KUKA KRL program: MyProgram_200().src

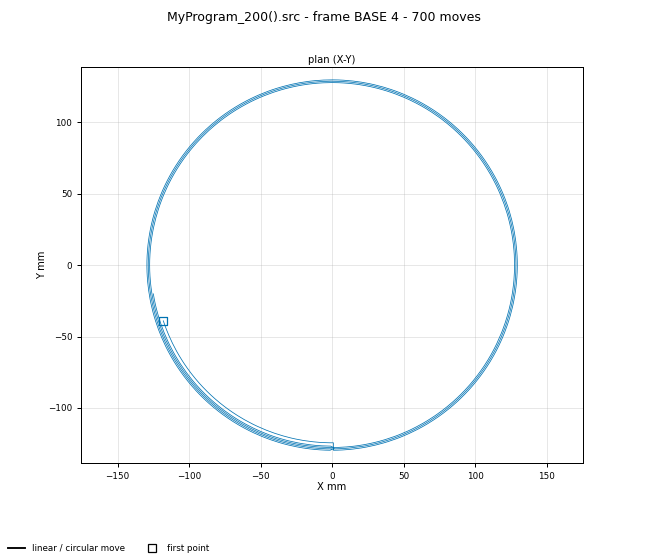
[picture p0: tool path of MyProgram_200().src in frame BASE 4, 700 of 700 moves have a stored position in this frame; points joined in program order, loops and branches not executed]
&ACCESS RVP
&REL 1
&PARAM TEMPLATE = C:\KRC\Roboter\Template\vorgabe
&PARAM EDITMASK = *
DEF MyProgram_200()
; ---- Setting reference (Base) ----
$BASE = BASE_DATA[4]

; --------------------------
; ---- Setting tool (TCP) ----
$TOOL = TOOL_DATA[3]
; --------------------------

$VEL.CP = VEL_APROX_PRINT
Startdeposition()
$VEL.CP = VEL_PRINT
LIN {X -118.0723,Y -39.0089,Z 143,A -163.9412,B 21.6303,C -0.9497,E1 21.4984,E2 611.217} C_DIS
LIN {X -116.9975,Y -42.1221,Z 143,A -162.4124,B 21.6305,C -0.9457,E1 21.4998,E2 609.6889} C_DIS
LIN {X -115.7317,Y -45.4869,Z 143,A -160.5818,B 21.6305,C -0.9476,E1 21.5017,E2 607.8411} C_DIS
LIN {X -114.1935,Y -49.2192,Z 143,A -158.8658,B 21.6309,C -0.9367,E1 21.5035,E2 606.1436} C_DIS
LIN {X -112.9502,Y -52.0092,Z 143,A -157.5422,B 21.6312,C -0.9295,E1 21.5051,E2 604.831} C_DIS
LIN {X -111.6598,Y -54.7252,Z 143,A -155.9756,B 21.631,C -0.9327,E1 21.507,E2 603.2459} C_DIS
LIN {X -110.264,Y -57.486,Z 143,A -154.672,B 21.6314,C -0.9241,E1 21.5086,E2 601.9576} C_DIS
LIN {X -108.8242,Y -60.1699,Z 143,A -153.2851,B 21.6316,C -0.9196,E1 21.5105,E2 600.5743} C_DIS
LIN {X -107.0458,Y -63.2806,Z 143,A -151.5187,B 21.6316,C -0.9197,E1 21.513,E2 598.7968} C_DIS
LIN {X -104.9264,Y -66.736,Z 143,A -149.6994,B 21.6318,C -0.913,E1 21.5156,E2 596.9849} C_DIS
LIN {X -103.3886,Y -69.0936,Z 143,A -148.3196,B 21.6318,C -0.913,E1 21.5178,E2 595.5972} C_DIS
LIN {X -101.1506,Y -72.3303,Z 143,A -146.4144,B 21.6318,C -0.912,E1 21.5208,E2 593.6835} C_DIS
LIN {X -98.5052,Y -75.8944,Z 143,A -144.3224,B 21.632,C -0.9089,E1 21.5244,E2 591.5883} C_DIS
LIN {X -95.4814,Y -79.6651,Z 143,A -142.1236,B 21.6323,C -0.9026,E1 21.5283,E2 589.3946} C_DIS
LIN {X -92.7275,Y -82.8538,Z 143,A -140.2642,B 21.6326,C -0.895,E1 21.5317,E2 587.5462} C_DIS
LIN {X -90.4998,Y -85.2814,Z 143,A -138.6409,B 21.6326,C -0.8958,E1 21.5348,E2 585.9122} C_DIS
LIN {X -87.3908,Y -88.4652,Z 143,A -136.6816,B 21.6328,C -0.8878,E1 21.5386,E2 583.9648} C_DIS
LIN {X -84.5496,Y -91.1842,Z 143,A -134.7498,B 21.6328,C -0.8889,E1 21.5425,E2 582.0209} C_DIS
LIN {X -81.7041,Y -93.7421,Z 143,A -132.9762,B 21.6329,C -0.8859,E1 21.5463,E2 580.2472} C_DIS
LIN {X -78.2894,Y -96.6125,Z 143,A -130.895,B 21.633,C -0.8831,E1 21.5507,E2 578.1644} C_DIS
LIN {X -75.1041,Y -99.1088,Z 143,A -129.1612,B 21.6334,C -0.8745,E1 21.5545,E2 576.4465} C_DIS
LIN {X -72.66,Y -100.9148,Z 143,A -127.794,B 21.6334,C -0.8708,E1 21.5576,E2 575.0838} C_DIS
LIN {X -69.8722,Y -102.8642,Z 143,A -126.1244,B 21.6334,C -0.8723,E1 21.5615,E2 573.4034} C_DIS
LIN {X -66.3215,Y -105.1883,Z 143,A -124.2918,B 21.6337,C -0.8644,E1 21.5658,E2 571.5855} C_DIS
LIN {X -63.9198,Y -106.6652,Z 143,A -122.8675,B 21.6337,C -0.8675,E1 21.5692,E2 570.1476} C_DIS
LIN {X -61.2916,Y -108.1971,Z 143,A -121.5152,B 21.6337,C -0.8635,E1 21.5724,E2 568.8014} C_DIS
LIN {X -58.1603,Y -109.9099,Z 143,A -119.9844,B 21.634,C -0.8567,E1 21.5762,E2 567.2839} C_DIS
LIN {X -55.5007,Y -111.2772,Z 143,A -118.5783,B 21.634,C -0.8561,E1 21.5797,E2 565.875} C_DIS
LIN {X -52.295,Y -112.818,Z 143,A -116.7434,B 21.6338,C -0.8622,E1 21.5844,E2 564.0183} C_DIS
LIN {X -48.773,Y -114.3864,Z 143,A -115.0584,B 21.634,C -0.8565,E1 21.5887,E2 562.344} C_DIS
LIN {X -46.1695,Y -115.4607,Z 143,A -113.7595,B 21.634,C -0.8553,E1 21.592,E2 561.045} C_DIS
LIN {X -42.8553,Y -116.7331,Z 143,A -112.1391,B 21.6342,C -0.8531,E1 21.5962,E2 559.4267} C_DIS
LIN {X -40.2291,Y -117.663,Z 143,A -110.8366,B 21.6342,C -0.8528,E1 21.5997,E2 558.1221} C_DIS
LIN {X -37.3375,Y -118.6123,Z 143,A -109.4335,B 21.6342,C -0.8517,E1 21.6034,E2 556.7188} C_DIS
LIN {X -34.4074,Y -119.4953,Z 143,A -107.8623,B 21.634,C -0.8574,E1 21.6077,E2 555.1293} C_DIS
LIN {X -31.4493,Y -120.308,Z 143,A -106.6081,B 21.6343,C -0.8499,E1 21.611,E2 553.8931} C_DIS
LIN {X -28.7309,Y -120.9852,Z 143,A -105.1465,B 21.634,C -0.8563,E1 21.615,E2 552.4119} C_DIS
LIN {X -25.5148,Y -121.7056,Z 143,A -103.8017,B 21.6343,C -0.8483,E1 21.6187,E2 551.0867} C_DIS
LIN {X -22.5042,Y -122.2974,Z 143,A -102.4392,B 21.6344,C -0.8457,E1 21.6224,E2 549.7297} C_DIS
LIN {X -19.7621,Y -122.7709,Z 143,A -100.9999,B 21.6342,C -0.8518,E1 21.6264,E2 548.2723} C_DIS
LIN {X -16.4893,Y -123.2516,Z 143,A -99.561,B 21.6344,C -0.8479,E1 21.6303,E2 546.8426} C_DIS
LIN {X -13.4636,Y -123.6184,Z 143,A -98.0599,B 21.6342,C -0.8517,E1 21.6345,E2 545.33} C_DIS
LIN {X -9.1471,Y -124.0125,Z 143,A -96.1214,B 21.6343,C -0.8491,E1 21.6399,E2 543.3975} C_DIS
LIN {X -6.1048,Y -124.1995,Z 143,A -94.6619,B 21.6343,C -0.8515,E1 21.644,E2 541.9311} C_DIS
LIN {X -1.7728,Y -124.3372,Z 143,A -92.7583,B 21.6343,C -0.8478,E1 21.6493,E2 540.0373} C_DIS
LIN {X 0.8945,Y -124.3442,Z 143,A -91.812,B 21.6348,C -0.8362,E1 21.6519,E2 539.1225} C_DIS
Enddeposition()
LIN {X 0.9181,Y -129.5582,Z 144,A -92.8615,B 24.9662,C -1.343,E1 25.0012,E2 539.3196} C_DIS
Startdeposition()
$VEL.CP = VEL_PRINT
LIN {X 3.5225,Y -129.5134,Z 144,A -91.2883,B 24.9651,C -1.3649,E1 25.0058,E2 537.6948} C_DIS
LIN {X 7.2346,Y -129.3611,Z 144,A -89.5433,B 24.9648,C -1.3708,E1 25.0106,E2 535.9365} C_DIS
LIN {X 11.6418,Y -129.0392,Z 144,A -87.6424,B 24.9648,C -1.369,E1 25.0159,E2 534.0408} C_DIS
LIN {X 14.6034,Y -128.7377,Z 144,A -86.2643,B 24.9647,C -1.373,E1 25.0198,E2 532.6543} C_DIS
LIN {X 18.1986,Y -128.2767,Z 144,A -84.9125,B 24.9653,C -1.3611,E1 25.0234,E2 531.3318} C_DIS
LIN {X 20.5727,Y -127.9195,Z 144,A -83.6159,B 24.9646,C -1.374,E1 25.0271,E2 530.0059} C_DIS
LIN {X 23.8922,Y -127.3398,Z 144,A -82.2252,B 24.9648,C -1.3701,E1 25.0309,E2 528.626} C_DIS
LIN {X 27.0969,Y -126.696,Z 144,A -80.8326,B 24.9649,C -1.3686,E1 25.0347,E2 527.2386} C_DIS
LIN {X 30.1007,Y -126.0161,Z 144,A -79.573,B 24.9651,C -1.3647,E1 25.0381,E2 525.9902} C_DIS
LIN {X 33.0736,Y -125.2688,Z 144,A -78.1067,B 24.9647,C -1.3718,E1 25.0421,E2 524.5091} C_DIS
LIN {X 36.068,Y -124.4397,Z 144,A -76.6892,B 24.9646,C -1.3756,E1 25.0459,E2 523.085} C_DIS
LIN {X 38.9883,Y -123.5562,Z 144,A -75.3211,B 24.9644,C -1.3782,E1 25.0496,E2 521.7132} C_DIS
LIN {X 42.2889,Y -122.465,Z 144,A -73.8532,B 24.9645,C -1.3766,E1 25.0534,E2 520.2521} C_DIS
LIN {X 45.0551,Y -121.4752,Z 144,A -72.5662,B 24.9645,C -1.3777,E1 25.0568,E2 518.9651} C_DIS
LIN {X 47.9955,Y -120.3439,Z 144,A -71.099,B 24.9641,C -1.3836,E1 25.0606,E2 517.4874} C_DIS
LIN {X 51.039,Y -119.0848,Z 144,A -69.8702,B 24.9646,C -1.3738,E1 25.0637,E2 516.2846} C_DIS
LIN {X 53.7433,Y -117.8903,Z 144,A -68.3328,B 24.9639,C -1.3879,E1 25.0677,E2 514.7175} C_DIS
LIN {X 56.9736,Y -116.3621,Z 144,A -66.8601,B 24.9641,C -1.3848,E1 25.0714,E2 513.256} C_DIS
LIN {X 59.5077,Y -115.089,Z 144,A -65.5363,B 24.9638,C -1.3906,E1 25.0747,E2 511.9222} C_DIS
LIN {X 63.1225,Y -113.1468,Z 144,A -63.6353,B 24.9634,C -1.3984,E1 25.0794,E2 510.0082} C_DIS
LIN {X 66.8503,Y -110.9845,Z 144,A -61.7577,B 24.9633,C -1.4005,E1 25.0839,E2 508.1314} C_DIS
LIN {X 70.7723,Y -108.5257,Z 144,A -59.7672,B 24.9633,C -1.4016,E1 25.0886,E2 506.1449} C_DIS
LIN {X 74.3388,Y -106.115,Z 144,A -57.7977,B 24.9628,C -1.409,E1 25.0931,E2 504.1646} C_DIS
LIN {X 77.8522,Y -103.5643,Z 144,A -55.9047,B 24.9627,C -1.4117,E1 25.0974,E2 502.272} C_DIS
LIN {X 81.2464,Y -100.9232,Z 144,A -54.0398,B 24.9625,C -1.4139,E1 25.1015,E2 500.4087} C_DIS
LIN {X 84.6421,Y -98.0928,Z 144,A -52.0954,B 24.9623,C -1.4179,E1 25.1056,E2 498.4625} C_DIS
LIN {X 87.5024,Y -95.5503,Z 144,A -50.5003,B 24.9624,C -1.4167,E1 25.1089,E2 496.8766} C_DIS
LIN {X 89.9458,Y -93.2538,Z 144,A -49.0251,B 24.9622,C -1.4199,E1 25.1119,E2 495.3999} C_DIS
LIN {X 92.7264,Y -90.4897,Z 144,A -47.2205,B 24.9618,C -1.4281,E1 25.1155,E2 493.5839} C_DIS
LIN {X 95.6696,Y -87.3727,Z 144,A -45.3787,B 24.9617,C -1.43,E1 25.119,E2 491.7455} C_DIS
LIN {X 98.2141,Y -84.5013,Z 144,A -43.6755,B 24.9614,C -1.4349,E1 25.1221,E2 490.0385} C_DIS
LIN {X 101.0014,Y -81.1495,Z 144,A -41.7257,B 24.9611,C -1.4412,E1 25.1255,E2 488.0827} C_DIS
LIN {X 103.67,Y -77.7122,Z 144,A -39.7722,B 24.9607,C -1.4481,E1 25.1289,E2 486.1222} C_DIS
LIN {X 106.115,Y -74.3388,Z 144,A -38.0216,B 24.9607,C -1.4484,E1 25.1317,E2 484.3797} C_DIS
LIN {X 108.4439,Y -70.8983,Z 144,A -36.1051,B 24.9602,C -1.4579,E1 25.1347,E2 482.4501} C_DIS
LIN {X 110.744,Y -67.2479,Z 144,A -34.2298,B 24.96,C -1.4617,E1 25.1374,E2 480.5754} C_DIS
LIN {X 113.0302,Y -63.3299,Z 144,A -32.3237,B 24.96,C -1.4623,E1 25.14,E2 478.6778} C_DIS
LIN {X 114.8245,Y -60.0114,Z 144,A -30.6729,B 24.9597,C -1.4664,E1 25.1422,E2 477.026} C_DIS
LIN {X 116.7251,Y -56.2264,Z 144,A -28.8572,B 24.9596,C -1.469,E1 25.1445,E2 475.2138} C_DIS
LIN {X 118.1717,Y -53.1176,Z 144,A -27.4238,B 24.9596,C -1.4692,E1 25.1461,E2 473.7877} C_DIS
LIN {X 119.4164,Y -50.2578,Z 144,A -25.9378,B 24.959,C -1.4793,E1 25.1478,E2 472.2861} C_DIS
LIN {X 120.6956,Y -47.1021,Z 144,A -24.5199,B 24.959,C -1.4793,E1 25.1492,E2 470.876} C_DIS
LIN {X 121.7925,Y -44.1889,Z 144,A -23.1418,B 24.9588,C -1.4837,E1 25.1506,E2 469.4952} C_DIS
LIN {X 122.6738,Y -41.6868,Z 144,A -21.8502,B 24.9582,C -1.4939,E1 25.1517,E2 468.1869} C_DIS
LIN {X 123.7738,Y -38.2914,Z 144,A -20.3604,B 24.9582,C -1.4942,E1 25.153,E2 466.7049} C_DIS
LIN {X 124.6622,Y -35.292,Z 144,A -19.0179,B 24.958,C -1.4964,E1 25.154,E2 465.3648} C_DIS
LIN {X 125.5247,Y -32.0878,Z 144,A -17.628,B 24.958,C -1.497,E1 25.155,E2 463.9816} C_DIS
LIN {X 126.2381,Y -29.1564,Z 144,A -16.2303,B 24.9576,C -1.5048,E1 25.1559,E2 462.5736} C_DIS
LIN {X 126.8882,Y -26.1835,Z 144,A -14.8491,B 24.9572,C -1.5111,E1 25.1567,E2 461.1856} C_DIS
LIN {X 127.5337,Y -22.83,Z 144,A -13.5152,B 24.9575,C -1.5065,E1 25.1574,E2 459.8703} C_DIS
LIN {X 128.1963,Y -18.7611,Z 144,A -11.7107,B 24.9572,C -1.5115,E1 25.1582,E2 458.0647} C_DIS
LIN {X 128.6178,Y -15.6082,Z 144,A -10.1493,B 24.9565,C -1.5245,E1 25.1588,E2 456.4818} C_DIS
LIN {X 128.9706,Y -12.3558,Z 144,A -8.7321,B 24.9563,C -1.5277,E1 25.1592,E2 455.0655} C_DIS
LIN {X 129.2709,Y -8.6987,Z 144,A -7.1495,B 24.9561,C -1.5309,E1 25.1595,E2 453.4848} C_DIS
LIN {X 129.4556,Y -5.2345,Z 144,A -5.5744,B 24.9557,C -1.5382,E1 25.1597,E2 451.9018} C_DIS
LIN {X 129.5553,Y -1.4347,Z 144,A -3.8664,B 24.9553,C -1.5452,E1 25.1597,E2 450.1875} C_DIS
LIN {X 129.5314,Y 2.8758,Z 144,A -2.0671,B 24.9553,C -1.5457,E1 25.1597,E2 448.3978} C_DIS
LIN {X 129.4093,Y 6.2771,Z 144,A -0.5027,B 24.9548,C -1.5539,E1 25.1595,E2 446.8234} C_DIS
LIN {X 129.1863,Y 9.8589,Z 144,A 1.0308,B 24.9546,C -1.5561,E1 25.1592,E2 445.2935} C_DIS
LIN {X 128.8637,Y 13.4323,Z 144,A 2.4842,B 24.9547,C -1.5541,E1 25.1589,E2 443.8536} C_DIS
LIN {X 128.5192,Y 16.4039,Z 144,A 3.7803,B 24.9546,C -1.557,E1 25.1584,E2 442.5584} C_DIS
LIN {X 128.1026,Y 19.3902,Z 144,A 5.3146,B 24.9537,C -1.5721,E1 25.1578,E2 440.9974} C_DIS
LIN {X 127.5895,Y 22.5183,Z 144,A 6.637,B 24.9537,C -1.5723,E1 25.1572,E2 439.6822} C_DIS
LIN {X 126.9963,Y 25.6519,Z 144,A 8.0598,B 24.9534,C -1.5775,E1 25.1564,E2 438.2555} C_DIS
LIN {X 126.307,Y 28.8547,Z 144,A 9.4009,B 24.9534,C -1.5763,E1 25.1556,E2 436.9251} C_DIS
LIN {X 125.6564,Y 31.5688,Z 144,A 10.7092,B 24.953,C -1.5842,E1 25.1547,E2 435.6057} C_DIS
LIN {X 124.8548,Y 34.6036,Z 144,A 12.1127,B 24.9527,C -1.5894,E1 25.1537,E2 434.1981} C_DIS
LIN {X 123.9722,Y 37.643,Z 144,A 13.4206,B 24.9527,C -1.5888,E1 25.1527,E2 432.8992} C_DIS
LIN {X 123.0062,Y 40.6885,Z 144,A 14.832,B 24.9525,C -1.593,E1 25.1515,E2 431.4857} C_DIS
LIN {X 121.9736,Y 43.6866,Z 144,A 16.3009,B 24.952,C -1.6009,E1 25.1501,E2 430.0065} C_DIS
LIN {X 120.8844,Y 46.6164,Z 144,A 17.5569,B 24.9521,C -1.5982,E1 25.1489,E2 428.7637} C_DIS
LIN {X 119.6862,Y 49.6117,Z 144,A 19.0301,B 24.9517,C -1.605,E1 25.1473,E2 427.2828} C_DIS
LIN {X 118.3697,Y 52.6751,Z 144,A 20.5347,B 24.9514,C -1.6109,E1 25.1456,E2 425.7724} C_DIS
LIN {X 116.984,Y 55.6845,Z 144,A 21.82,B 24.9517,C -1.6056,E1 25.1441,E2 424.5067} C_DIS
LIN {X 115.5871,Y 58.5292,Z 144,A 23.3224,B 24.9511,C -1.615,E1 25.1422,E2 422.9902} C_DIS
LIN {X 113.9385,Y 61.682,Z 144,A 25.0888,B 24.9502,C -1.6297,E1 25.1399,E2 421.1983} C_DIS
LIN {X 111.8345,Y 65.4184,Z 144,A 26.957,B 24.95,C -1.6334,E1 25.1373,E2 419.331} C_DIS
LIN {X 109.4219,Y 69.3785,Z 144,A 28.9822,B 24.9498,C -1.6376,E1 25.1343,E2 417.3062} C_DIS
LIN {X 107.0606,Y 72.9703,Z 144,A 30.9092,B 24.9494,C -1.6439,E1 25.1313,E2 415.3738} C_DIS
LIN {X 104.5579,Y 76.5125,Z 144,A 32.7988,B 24.9491,C -1.6473,E1 25.1282,E2 413.4854} C_DIS
LIN {X 102.0399,Y 79.8397,Z 144,A 34.6354,B 24.9489,C -1.6515,E1 25.1251,E2 411.6477} C_DIS
LIN {X 99.1372,Y 83.4166,Z 144,A 36.6214,B 24.9488,C -1.6537,E1 25.1215,E2 409.6656} C_DIS
LIN {X 96.6742,Y 86.2591,Z 144,A 38.1982,B 24.9488,C -1.653,E1 25.1187,E2 408.0976} C_DIS
LIN {X 94.1055,Y 89.0543,Z 144,A 39.8981,B 24.9485,C -1.6579,E1 25.1154,E2 406.3935} C_DIS
LIN {X 91.1558,Y 92.0714,Z 144,A 41.7621,B 24.9482,C -1.6619,E1 25.1117,E2 404.528} C_DIS
LIN {X 88.1187,Y 94.9822,Z 144,A 43.6758,B 24.9478,C -1.6686,E1 25.1078,E2 402.6062} C_DIS
LIN {X 84.8691,Y 97.8973,Z 144,A 45.5005,B 24.9479,C -1.667,E1 25.104,E2 400.7927} C_DIS
LIN {X 81.7997,Y 100.4756,Z 144,A 47.3562,B 24.9474,C -1.6748,E1 25.1,E2 398.9256} C_DIS
LIN {X 78.3783,Y 103.1673,Z 144,A 49.3219,B 24.9471,C -1.6805,E1 25.0957,E2 396.9537} C_DIS
LIN {X 74.876,Y 105.7361,Z 144,A 51.2149,B 24.947,C -1.6824,E1 25.0914,E2 395.0628} C_DIS
LIN {X 71.0441,Y 108.3479,Z 144,A 53.2303,B 24.9469,C -1.684,E1 25.0867,E2 393.0504} C_DIS
LIN {X 67.3967,Y 110.6541,Z 144,A 55.1766,B 24.9465,C -1.6889,E1 25.0821,E2 391.0986} C_DIS
LIN {X 63.689,Y 112.8284,Z 144,A 57.0503,B 24.9465,C -1.6903,E1 25.0775,E2 389.2272} C_DIS
LIN {X 59.7209,Y 114.977,Z 144,A 59.0445,B 24.9463,C -1.693,E1 25.0726,E2 387.2323} C_DIS
LIN {X 56.0887,Y 116.7909,Z 144,A 60.7162,B 24.9465,C -1.6889,E1 25.0685,E2 385.5748} C_DIS
LIN {X 53.1708,Y 118.148,Z 144,A 61.925,B 24.9471,C -1.6796,E1 25.0655,E2 384.391} C_DIS
LIN {X 50.3192,Y 119.3907,Z 144,A 63.4841,B 24.9464,C -1.6905,E1 25.0614,E2 382.8098} C_DIS
LIN {X 47.2157,Y 120.6514,Z 144,A 64.9763,B 24.9464,C -1.6926,E1 25.0575,E2 381.316} C_DIS
LIN {X 44.2201,Y 121.7813,Z 144,A 66.378,B 24.9463,C -1.6932,E1 25.0539,E2 379.9158} C_DIS
LIN {X 41.2103,Y 122.8324,Z 144,A 67.594,B 24.9468,C -1.6846,E1 25.0507,E2 378.7227} C_DIS
LIN {X 38.1472,Y 123.8179,Z 144,A 69.2154,B 24.9461,C -1.6958,E1 25.0463,E2 377.0776} C_DIS
LIN {X 35.483,Y 124.6088,Z 144,A 70.5267,B 24.9458,C -1.7009,E1 25.0428,E2 375.7565} C_DIS
LIN {X 32.3099,Y 125.4684,Z 144,A 71.9309,B 24.9458,C -1.6993,E1 25.039,E2 374.3582} C_DIS
LIN {X 29.3998,Y 126.1825,Z 144,A 73.296,B 24.9458,C -1.7021,E1 25.0353,E2 372.9885} C_DIS
LIN {X 26.0384,Y 126.9177,Z 144,A 74.76,B 24.9458,C -1.6999,E1 25.0313,E2 371.5315} C_DIS
LIN {X 22.9002,Y 127.5212,Z 144,A 76.0299,B 24.9463,C -1.6933,E1 25.0279,E2 370.2788} C_DIS
LIN {X 20.5727,Y 127.9195,Z 144,A 77.2797,B 24.9456,C -1.704,E1 25.0244,E2 369.005} C_DIS
LIN {X 17.5811,Y 128.3649,Z 144,A 78.6134,B 24.9456,C -1.7041,E1 25.0207,E2 367.672} C_DIS
LIN {X 14.6034,Y 128.7377,Z 144,A 80.0011,B 24.9454,C -1.7074,E1 25.0168,E2 366.2776} C_DIS
LIN {X 10.9979,Y 129.0936,Z 144,A 81.3371,B 24.9462,C -1.6942,E1 25.0132,E2 364.9735} C_DIS
LIN {X 8.0925,Y 129.3083,Z 144,A 82.7577,B 24.9458,C -1.7009,E1 25.0092,E2 363.5378} C_DIS
LIN {X 4.3229,Y 129.4911,Z 144,A 84.5434,B 24.9454,C -1.7066,E1 25.0042,E2 361.739} C_DIS
LIN {X 0.5242,Y 129.5604,Z 144,A 86.1196,B 24.9458,C -1.7012,E1 24.9998,E2 360.1759} C_DIS
LIN {X -3.1801,Y 129.5229,Z 144,A 87.5856,B 24.9463,C -1.6922,E1 24.9958,E2 358.7312} C_DIS
LIN {X -6.0827,Y 129.4191,Z 144,A 88.8724,B 24.9463,C -1.6919,E1 24.9922,E2 357.4448} C_DIS
LIN {X -9.324,Y 129.2253,Z 144,A 90.2842,B 24.9465,C -1.6901,E1 24.9883,E2 356.0368} C_DIS
LIN {X -12.2468,Y 128.9811,Z 144,A 91.6532,B 24.9463,C -1.693,E1 24.9844,E2 354.6602} C_DIS
LIN {X -16.4039,Y 128.5192,Z 144,A 93.6229,B 24.946,C -1.6979,E1 24.9789,E2 352.6777} C_DIS
LIN {X -19.5971,Y 128.0706,Z 144,A 94.9456,B 24.9464,C -1.6918,E1 24.9753,E2 351.3682} C_DIS
LIN {X -22.7107,Y 127.5551,Z 144,A 96.3497,B 24.9464,C -1.6912,E1 24.9714,E2 349.9642} C_DIS
LIN {X -25.615,Y 127.0038,Z 144,A 97.7365,B 24.9462,C -1.6941,E1 24.9676,E2 348.5692} C_DIS
LIN {X -28.6159,Y 126.3615,Z 144,A 99.0325,B 24.9465,C -1.6898,E1 24.9641,E2 347.2815} C_DIS
LIN {X -31.4943,Y 125.6754,Z 144,A 100.4585,B 24.9462,C -1.6943,E1 24.9602,E2 345.843} C_DIS
LIN {X -34.6092,Y 124.8532,Z 144,A 101.8797,B 24.9463,C -1.6927,E1 24.9564,E2 344.4235} C_DIS
LIN {X -38.9883,Y 123.5562,Z 144,A 103.8983,B 24.9465,C -1.6903,E1 24.951,E2 342.4071} C_DIS
LIN {X -42.0033,Y 122.564,Z 144,A 105.1415,B 24.9471,C -1.6807,E1 24.9478,E2 341.1843} C_DIS
LIN {X -45.0101,Y 121.492,Z 144,A 106.7288,B 24.9466,C -1.6874,E1 24.9435,E2 339.5778} C_DIS
LIN {X -48.084,Y 120.3082,Z 144,A 108.1286,B 24.9469,C -1.6827,E1 24.9399,E2 338.1863} C_DIS
LIN {X -50.9868,Y 119.1073,Z 144,A 109.4465,B 24.9473,C -1.6772,E1 24.9366,E2 336.8785} C_DIS
LIN {X -53.8875,Y 117.8237,Z 144,A 110.9243,B 24.9472,C -1.6786,E1 24.9328,E2 335.3936} C_DIS
LIN {X -56.8988,Y 116.399,Z 144,A 112.4837,B 24.9471,C -1.6805,E1 24.9288,E2 333.8258} C_DIS
LIN {X -59.8483,Y 114.9102,Z 144,A 113.9527,B 24.9472,C -1.6784,E1 24.9252,E2 332.3577} C_DIS
LIN {X -63.689,Y 112.8284,Z 144,A 115.9154,B 24.9473,C -1.6765,E1 24.9204,E2 330.3941} C_DIS
LIN {X -67.3967,Y 110.6541,Z 144,A 117.8831,B 24.9473,C -1.6761,E1 24.9157,E2 328.4211} C_DIS
LIN {X -71.0441,Y 108.3479,Z 144,A 119.7942,B 24.9476,C -1.6726,E1 24.9112,E2 326.5124} C_DIS
LIN {X -74.876,Y 105.7361,Z 144,A 121.8118,B 24.9479,C -1.6668,E1 24.9066,E2 324.5016} C_DIS
LIN {X -78.3839,Y 103.163,Z 144,A 123.7133,B 24.9483,C -1.6616,E1 24.9023,E2 322.6056} C_DIS
LIN {X -81.6635,Y 100.5869,Z 144,A 125.6622,B 24.9483,C -1.6626,E1 24.898,E2 320.6472} C_DIS
LIN {X -85.0895,Y 97.705,Z 144,A 127.6055,B 24.9486,C -1.6563,E1 24.8939,E2 318.7113} C_DIS
LIN {X -88.4135,Y 94.7077,Z 144,A 129.5845,B 24.9489,C -1.6516,E1 24.8899,E2 316.7355} C_DIS
LIN {X -91.1453,Y 92.0818,Z 144,A 131.1857,B 24.9494,C -1.6439,E1 24.8867,E2 315.1458} C_DIS
LIN {X -93.8339,Y 89.3405,Z 144,A 132.9675,B 24.9494,C -1.6437,E1 24.8832,E2 313.3569} C_DIS
LIN {X -96.7917,Y 86.1278,Z 144,A 134.8818,B 24.9497,C -1.6379,E1 24.8796,E2 311.4479} C_DIS
LIN {X -99.4108,Y 83.0904,Z 144,A 136.6399,B 24.9501,C -1.6325,E1 24.8765,E2 309.6947} C_DIS
LIN {X -102.0399,Y 79.8397,Z 144,A 138.4989,B 24.9503,C -1.628,E1 24.8732,E2 307.8377} C_DIS
LIN {X -104.5579,Y 76.5125,Z 144,A 140.4014,B 24.9505,C -1.6256,E1 24.8701,E2 305.9317} C_DIS
LIN {X -107.0606,Y 72.9703,Z 144,A 142.4005,B 24.9505,C -1.624,E1 24.8669,E2 303.9264} C_DIS
LIN {X -109.3662,Y 69.4669,Z 144,A 144.2397,B 24.9509,C -1.6179,E1 24.8641,E2 302.0924} C_DIS
LIN {X -111.5045,Y 65.9802,Z 144,A 146.0125,B 24.9514,C -1.6109,E1 24.8616,E2 300.3272} C_DIS
LIN {X -113.5451,Y 62.4032,Z 144,A 147.8887,B 24.9515,C -1.6081,E1 24.859,E2 298.4478} C_DIS
LIN {X -115.3418,Y 59.0112,Z 144,A 149.4956,B 24.9521,C -1.5988,E1 24.8569,E2 296.8546} C_DIS
LIN {X -116.7011,Y 56.2765,Z 144,A 150.8766,B 24.9523,C -1.5961,E1 24.8553,E2 295.4726} C_DIS
LIN {X -118.1615,Y 53.1404,Z 144,A 152.3308,B 24.9528,C -1.5878,E1 24.8536,E2 294.0301} C_DIS
LIN {X -119.4392,Y 50.2032,Z 144,A 153.7509,B 24.953,C -1.5836,E1 24.852,E2 292.6122} C_DIS
LIN {X -120.6774,Y 47.1489,Z 144,A 155.2693,B 24.9531,C -1.5819,E1 24.8504,E2 291.0894} C_DIS
LIN {X -121.7241,Y 44.3786,Z 144,A 156.4524,B 24.9537,C -1.5718,E1 24.8493,E2 289.9237} C_DIS
LIN {X -122.8274,Y 41.2255,Z 144,A 158.0637,B 24.9537,C -1.5734,E1 24.8478,E2 288.2993} C_DIS
LIN {X -123.7547,Y 38.3536,Z 144,A 159.4672,B 24.9537,C -1.5724,E1 24.8466,E2 286.8903} C_DIS
LIN {X -124.6157,Y 35.4584,Z 144,A 160.8017,B 24.9539,C -1.568,E1 24.8456,E2 285.5585} C_DIS
LIN {X -125.5074,Y 32.1561,Z 144,A 162.3194,B 24.9542,C -1.5634,E1 24.8445,E2 284.043} C_DIS
LIN {X -126.5646,Y 27.7052,Z 144,A 164.3096,B 24.9547,C -1.5552,E1 24.8433,E2 282.0606} C_DIS
LIN {X -127.2378,Y 24.4256,Z 144,A 165.8293,B 24.9549,C -1.5522,E1 24.8425,E2 280.539} C_DIS
LIN {X -127.824,Y 21.1455,Z 144,A 167.3512,B 24.955,C -1.5497,E1 24.8418,E2 279.0141} C_DIS
LIN {X -128.4071,Y 17.2593,Z 144,A 169.1103,B 24.9553,C -1.5449,E1 24.8411,E2 277.2558} C_DIS
LIN {X -128.8316,Y 13.7309,Z 144,A 170.6787,B 24.9556,C -1.5396,E1 24.8406,E2 275.6907} C_DIS
LIN {X -129.1998,Y 9.6732,Z 144,A 172.452,B 24.956,C -1.5323,E1 24.8402,E2 273.9242} C_DIS
LIN {X -129.3966,Y 6.529,Z 144,A 173.8462,B 24.9563,C -1.5278,E1 24.8399,E2 272.5324} C_DIS
LIN {X -129.5314,Y 2.8758,Z 144,A 175.6226,B 24.9561,C -1.5299,E1 24.8399,E2 270.7402} C_DIS
LIN {X -129.5586,Y -1.0172,Z 144,A 177.3382,B 24.9565,C -1.524,E1 24.8399,E2 269.0283} C_DIS
LIN {X -129.4697,Y -4.8731,Z 144,A 178.8924,B 24.9572,C -1.5113,E1 24.8399,E2 267.4951} C_DIS
LIN {X -129.3157,Y -7.9717,Z 144,A -179.6588,B 24.9572,C -1.5104,E1 24.8402,E2 266.0396} C_DIS
LIN {X -129.0124,Y -11.921,Z 144,A -177.8834,B 24.9575,C -1.5058,E1 24.8406,E2 264.2646} C_DIS
LIN {X -128.7048,Y -14.8785,Z 144,A -176.5345,B 24.9577,C -1.5031,E1 24.841,E2 262.914} C_DIS
LIN {X -128.3157,Y -17.9252,Z 144,A -175.2622,B 24.9581,C -1.4947,E1 24.8415,E2 261.6542} C_DIS
LIN {X -127.851,Y -20.9836,Z 144,A -173.8162,B 24.9581,C -1.494,E1 24.8421,E2 260.2013} C_DIS
LIN {X -127.3398,Y -23.8922,Z 144,A -172.5102,B 24.9584,C -1.4898,E1 24.8428,E2 258.8976} C_DIS
LIN {X -126.7769,Y -26.7223,Z 144,A -171.198,B 24.9586,C -1.4874,E1 24.8435,E2 257.5832} C_DIS
LIN {X -126.0588,Y -29.9236,Z 144,A -169.7544,B 24.9588,C -1.4825,E1 24.8444,E2 256.1429} C_DIS
LIN {X -125.3513,Y -32.7641,Z 144,A -168.421,B 24.9589,C -1.4803,E1 24.8453,E2 254.807} C_DIS
LIN {X -124.469,Y -35.9681,Z 144,A -167.1517,B 24.9597,C -1.4663,E1 24.8463,E2 253.5637} C_DIS
LIN {X -123.5562,Y -38.9883,Z 144,A -165.6131,B 24.9596,C -1.4687,E1 24.8476,E2 252.0104} C_DIS
LIN {X -122.5372,Y -42.0807,Z 144,A -164.3283,B 24.9602,C -1.457,E1 24.8487,E2 250.7462} C_DIS
LIN {X -121.492,Y -45.0101,Z 144,A -162.7481,B 24.9599,C -1.4625,E1 24.8502,E2 249.144} C_DIS
LIN {X -120.3001,Y -48.1043,Z 144,A -161.3162,B 24.9603,C -1.4565,E1 24.8517,E2 247.7183} C_DIS
LIN {X -119.1001,Y -51.0035,Z 144,A -159.9046,B 24.9604,C -1.4536,E1 24.8532,E2 246.3059} C_DIS
LIN {X -117.7214,Y -54.1086,Z 144,A -158.593,B 24.9611,C -1.4402,E1 24.8547,E2 245.0192} C_DIS
LIN {X -116.4101,Y -56.8763,Z 144,A -156.9625,B 24.9606,C -1.4494,E1 24.8567,E2 243.3579} C_DIS
LIN {X -114.972,Y -59.7306,Z 144,A -155.5189,B 24.9608,C -1.4468,E1 24.8585,E2 241.9127} C_DIS
LIN {X -112.8284,Y -63.689,Z 144,A -153.5272,B 24.9611,C -1.4413,E1 24.8612,E2 239.9236} C_DIS
LIN {X -110.6541,Y -67.3967,Z 144,A -151.5834,B 24.9613,C -1.4382,E1 24.864,E2 237.9771} C_DIS
LIN {X -108.4439,Y -70.8983,Z 144,A -149.6972,B 24.9613,C -1.436,E1 24.8669,E2 236.0866} C_DIS
LIN {X -106.1014,Y -74.358,Z 144,A -147.842,B 24.9616,C -1.4316,E1 24.8698,E2 234.2327} C_DIS
LIN {X -103.4888,Y -77.9522,Z 144,A -145.9135,B 24.962,C -1.4249,E1 24.873,E2 232.3108} C_DIS
LIN {X -101.0014,Y -81.1495,Z 144,A -144.0823,B 24.962,C -1.4224,E1 24.8762,E2 230.477} C_DIS
LIN {X -98.1176,Y -84.6133,Z 144,A -142.1096,B 24.9624,C -1.4167,E1 24.8797,E2 228.5088} C_DIS
LIN {X -95.23,Y -87.8508,Z 144,A -140.1747,B 24.9626,C -1.4131,E1 24.8834,E2 226.5739} C_DIS
LIN {X -92.2061,Y -91.0202,Z 144,A -138.1939,B 24.9627,C -1.411,E1 24.8872,E2 224.5897} C_DIS
LIN {X -89.213,Y -93.9557,Z 144,A -136.3566,B 24.963,C -1.4062,E1 24.8909,E2 222.7561} C_DIS
LIN {X -86.0382,Y -96.871,Z 144,A -134.4449,B 24.9631,C -1.4026,E1 24.8949,E2 220.8454} C_DIS
LIN {X -82.9556,Y -99.5239,Z 144,A -132.6022,B 24.9632,C -1.4012,E1 24.8988,E2 218.9987} C_DIS
LIN {X -79.5702,Y -102.2503,Z 144,A -130.6906,B 24.9634,C -1.3972,E1 24.903,E2 217.0898} C_DIS
LIN {X -76.1935,Y -104.7906,Z 144,A -128.8238,B 24.9636,C -1.3937,E1 24.9072,E2 215.2244} C_DIS
LIN {X -72.4461,Y -107.4154,Z 144,A -126.8364,B 24.9639,C -1.3886,E1 24.9117,E2 213.2427} C_DIS
LIN {X -68.8043,Y -109.7844,Z 144,A -124.8516,B 24.9639,C -1.3886,E1 24.9164,E2 211.2513} C_DIS
LIN {X -65.1188,Y -112.0093,Z 144,A -122.955,B 24.964,C -1.3855,E1 24.921,E2 209.3565} C_DIS
LIN {X -61.111,Y -114.2453,Z 144,A -120.9312,B 24.9642,C -1.3824,E1 24.9259,E2 207.3342} C_DIS
LIN {X -57.7122,Y -115.9977,Z 144,A -119.3095,B 24.9645,C -1.3768,E1 24.93,E2 205.7215} C_DIS
LIN {X -54.8054,Y -117.3992,Z 144,A -117.8564,B 24.9645,C -1.3764,E1 24.9336,E2 204.2656} C_DIS
LIN {X -51.6024,Y -118.8412,Z 144,A -116.4316,B 24.9649,C -1.3683,E1 24.9372,E2 202.8568} C_DIS
LIN {X -48.8578,Y -119.9963,Z 144,A -114.9784,B 24.9647,C -1.3737,E1 24.941,E2 201.3875} C_DIS
LIN {X -45.6778,Y -121.2419,Z 144,A -113.5957,B 24.9651,C -1.3659,E1 24.9446,E2 200.0204} C_DIS
LIN {X -43.1919,Y -122.152,Z 144,A -112.2657,B 24.9647,C -1.3727,E1 24.9481,E2 198.6714} C_DIS
LIN {X -39.6352,Y -123.3496,Z 144,A -110.7239,B 24.9651,C -1.3655,E1 24.9522,E2 197.1439} C_DIS
LIN {X -37.0099,Y -124.164,Z 144,A -109.3897,B 24.9648,C -1.3706,E1 24.9558,E2 195.7954} C_DIS
LIN {X -33.6508,Y -125.1149,Z 144,A -107.9453,B 24.9651,C -1.3646,E1 24.9596,E2 194.363} C_DIS
LIN {X -30.606,Y -125.8943,Z 144,A -106.5527,B 24.9651,C -1.3639,E1 24.9634,E2 192.9701} C_DIS
LIN {X -27.4507,Y -126.6196,Z 144,A -105.2144,B 24.9654,C -1.3585,E1 24.967,E2 191.6429} C_DIS
LIN {X -25.0807,Y -127.1126,Z 144,A -103.9444,B 24.9649,C -1.3681,E1 24.9706,E2 190.3487} C_DIS
LIN {X -21.7575,Y -127.7219,Z 144,A -102.511,B 24.9651,C -1.3645,E1 24.9745,E2 188.9223} C_DIS
LIN {X -18.4632,Y -128.2389,Z 144,A -101.0632,B 24.9652,C -1.3628,E1 24.9785,E2 187.4774} C_DIS
LIN {X -15.2487,Y -128.6607,Z 144,A -99.6054,B 24.9652,C -1.3638,E1 24.9825,E2 186.0163} C_DIS
LIN {X -11.3319,Y -129.0654,Z 144,A -97.8397,B 24.9652,C -1.3648,E1 24.9875,E2 184.2471} C_DIS
LIN {X -8.3908,Y -129.2899,Z 144,A -96.5122,B 24.965,C -1.366,E1 24.9912,E2 182.9163} C_DIS
LIN {X -4.7402,Y -129.4749,Z 144,A -94.8458,B 24.965,C -1.3687,E1 24.9958,E2 181.2431} C_DIS
LIN {X -1.4347,Y -129.5553,Z 144,A -93.441,B 24.965,C -1.366,E1 24.9997,E2 179.8447} C_DIS
LIN {X -1.4347,Y -129.5553,Z 144,A -93.441,B 24.965,C -1.366,E1 24.9997,E2 179.8447} C_DIS
Enddeposition()
LIN {X 0.9199,Y -128.5887,Z 144,A -93.2284,B 24.822,C -1.3109,E1 24.8545,E2 179.7433} C_DIS
Startdeposition()
$VEL.CP = VEL_PRINT
LIN {X -3.6308,Y -128.5472,Z 144,A -95.152,B 24.8218,C -1.3156,E1 24.8491,E2 181.6559} C_DIS
LIN {X -9.1432,Y -128.2732,Z 144,A -97.5729,B 24.8218,C -1.3173,E1 24.8424,E2 184.0733} C_DIS
LIN {X -12.2021,Y -128.0182,Z 144,A -99.2442,B 24.8225,C -1.3025,E1 24.8376,E2 185.781} C_DIS
LIN {X -17.1823,Y -127.4462,Z 144,A -102.184,B 24.8241,C -1.2685,E1 24.8293,E2 188.804} C_DIS
LIN {X -23.7565,Y -126.3855,Z 144,A -104.219,B 24.8219,C -1.3148,E1 24.824,E2 190.7306} C_DIS
LIN {X -27.1436,Y -125.7009,Z 144,A -105.7055,B 24.8217,C -1.3181,E1 24.8199,E2 192.2109} C_DIS
LIN {X -30.7997,Y -124.8573,Z 144,A -107.4985,B 24.8219,C -1.3131,E1 24.815,E2 194.0185} C_DIS
LIN {X -34.4965,Y -123.885,Z 144,A -109.0349,B 24.8215,C -1.3223,E1 24.8109,E2 195.5352} C_DIS
LIN {X -37.7046,Y -122.9465,Z 144,A -110.5756,B 24.8215,C -1.3209,E1 24.8068,E2 197.0819} C_DIS
LIN {X -41.2877,Y -121.7919,Z 144,A -112.2078,B 24.8214,C -1.3244,E1 24.8025,E2 198.7087} C_DIS
LIN {X -44.4075,Y -120.6896,Z 144,A -113.8416,B 24.8217,C -1.318,E1 24.7981,E2 200.3611} C_DIS
LIN {X -47.7918,Y -119.388,Z 144,A -115.3659,B 24.8214,C -1.324,E1 24.7942,E2 201.8743} C_DIS
LIN {X -50.5783,Y -118.235,Z 144,A -116.9023,B 24.8218,C -1.3162,E1 24.7902,E2 203.4331} C_DIS
LIN {X -55.1361,Y -116.179,Z 144,A -118.9431,B 24.8212,C -1.3278,E1 24.7851,E2 205.4512} C_DIS
LIN {X -57.9028,Y -114.8257,Z 144,A -120.4671,B 24.8215,C -1.3222,E1 24.7812,E2 206.9927} C_DIS
LIN {X -61.884,Y -112.7316,Z 144,A -122.4198,B 24.8212,C -1.3274,E1 24.7764,E2 208.9385} C_DIS
LIN {X -65.595,Y -110.6133,Z 144,A -124.3368,B 24.8212,C -1.3295,E1 24.7718,E2 210.8561} C_DIS
LIN {X -69.4465,Y -108.2364,Z 144,A -126.3218,B 24.8209,C -1.3342,E1 24.7671,E2 212.8363} C_DIS
LIN {X -73.0534,Y -105.8359,Z 144,A -128.2517,B 24.8207,C -1.3374,E1 24.7627,E2 214.7651} C_DIS
LIN {X -76.7246,Y -103.2049,Z 144,A -130.2857,B 24.8206,C -1.3399,E1 24.7581,E2 216.8003} C_DIS
LIN {X -80.0299,Y -100.6635,Z 144,A -132.0855,B 24.8203,C -1.3461,E1 24.7541,E2 218.592} C_DIS
LIN {X -83.1208,Y -98.1269,Z 144,A -133.969,B 24.8203,C -1.3447,E1 24.7501,E2 220.4861} C_DIS
LIN {X -86.5847,Y -95.0845,Z 144,A -136.0139,B 24.8201,C -1.3493,E1 24.7458,E2 222.5282} C_DIS
LIN {X -89.729,Y -92.1237,Z 144,A -137.9766,B 24.8201,C -1.3515,E1 24.7419,E2 224.4937} C_DIS
LIN {X -92.813,Y -89.0153,Z 144,A -139.9289,B 24.8198,C -1.3557,E1 24.7381,E2 226.4443} C_DIS
LIN {X -95.8004,Y -85.7916,Z 144,A -141.8163,B 24.8194,C -1.3635,E1 24.7345,E2 228.3215} C_DIS
LIN {X -98.4515,Y -82.7359,Z 144,A -143.6753,B 24.8194,C -1.3651,E1 24.7311,E2 230.1852} C_DIS
LIN {X -101.2678,Y -79.2641,Z 144,A -145.448,B 24.8185,C -1.3802,E1 24.7281,E2 231.9302} C_DIS
LIN {X -103.5549,Y -76.2517,Z 144,A -147.3513,B 24.8188,C -1.3742,E1 24.7249,E2 233.857} C_DIS
LIN {X -105.9046,Y -72.9532,Z 144,A -149.136,B 24.8186,C -1.3797,E1 24.722,E2 235.6373} C_DIS
LIN {X -108.4934,Y -69.045,Z 144,A -151.3174,B 24.8185,C -1.3809,E1 24.7187,E2 237.8269} C_DIS
LIN {X -110.73,Y -65.3978,Z 144,A -153.2405,B 24.8183,C -1.3853,E1 24.7159,E2 239.7496} C_DIS
LIN {X -112.3325,Y -62.6056,Z 144,A -154.8712,B 24.8185,C -1.3802,E1 24.7137,E2 241.4011} C_DIS
LIN {X -114.3606,Y -58.8164,Z 144,A -156.3643,B 24.8172,C -1.405,E1 24.7118,E2 242.8426} C_DIS
LIN {X -116.5619,Y -54.3222,Z 144,A -158.7063,B 24.8172,C -1.4062,E1 24.7089,E2 245.1946} C_DIS
LIN {X -117.9117,Y -51.3261,Z 144,A -160.229,B 24.8171,C -1.4078,E1 24.7072,E2 246.7219} C_DIS
LIN {X -119.2357,Y -48.1695,Z 144,A -161.7271,B 24.8168,C -1.4135,E1 24.7056,E2 248.2147} C_DIS
LIN {X -120.4363,Y -45.0837,Z 144,A -163.2399,B 24.8166,C -1.4162,E1 24.7041,E2 249.7296} C_DIS
LIN {X -121.7288,Y -41.4733,Z 144,A -165.123,B 24.8168,C -1.4134,E1 24.7023,E2 251.6303} C_DIS
LIN {X -122.9747,Y -37.6125,Z 144,A -166.8304,B 24.8162,C -1.4235,E1 24.7009,E2 253.3232} C_DIS
LIN {X -123.8421,Y -34.6498,Z 144,A -168.1875,B 24.816,C -1.4286,E1 24.6999,E2 254.676} C_DIS
LIN {X -124.8928,Y -30.6523,Z 144,A -170.0711,B 24.8158,C -1.4325,E1 24.6986,E2 256.5616} C_DIS
LIN {X -125.7042,Y -27.1283,Z 144,A -171.6353,B 24.8154,C -1.4397,E1 24.6976,E2 258.1176} C_DIS
LIN {X -126.4788,Y -23.2597,Z 144,A -173.486,B 24.8153,C -1.441,E1 24.6967,E2 259.9761} C_DIS
LIN {X -127.1137,Y -19.4849,Z 144,A -175.135,B 24.8148,C -1.4491,E1 24.6959,E2 261.6156} C_DIS
LIN {X -127.6545,Y -15.5556,Z 144,A -176.9398,B 24.8146,C -1.4531,E1 24.6953,E2 263.4218} C_DIS
LIN {X -128.06,Y -11.7666,Z 144,A -178.7198,B 24.8146,C -1.4549,E1 24.6948,E2 265.2084} C_DIS
LIN {X -128.3689,Y -7.6837,Z 144,A 179.5114,B 24.8141,C -1.4634,E1 24.6945,E2 266.9675} C_DIS
LIN {X -128.5464,Y -3.6615,Z 144,A 177.7346,B 24.8137,C -1.47,E1 24.6943,E2 268.7391} C_DIS
LIN {X -128.6002,Y 0.3582,Z 144,A 175.8104,B 24.8137,C -1.4698,E1 24.6943,E2 270.6754} C_DIS
LIN {X -128.5117,Y 4.7322,Z 144,A 173.9676,B 24.8131,C -1.4811,E1 24.6943,E2 272.5024} C_DIS
LIN {X -128.3154,Y 8.5521,Z 144,A 172.1484,B 24.8131,C -1.4814,E1 24.6947,E2 274.3318} C_DIS
LIN {X -128.0027,Y 12.3639,Z 144,A 170.5339,B 24.8125,C -1.4911,E1 24.6951,E2 275.9327} C_DIS
LIN {X -127.5597,Y 16.3162,Z 144,A 168.703,B 24.8123,C -1.4943,E1 24.6957,E2 277.7672} C_DIS
LIN {X -127.0249,Y 20.0583,Z 144,A 166.9904,B 24.8121,C -1.4985,E1 24.6964,E2 279.4799} C_DIS
LIN {X -126.3285,Y 24.0545,Z 144,A 165.2542,B 24.8116,C -1.5077,E1 24.6973,E2 281.2045} C_DIS
LIN {X -125.6638,Y 27.3155,Z 144,A 163.9083,B 24.8109,C -1.5187,E1 24.698,E2 282.5319} C_DIS
LIN {X -124.5553,Y 31.9937,Z 144,A 161.4788,B 24.8113,C -1.5126,E1 24.6997,E2 284.9905} C_DIS
LIN {X -123.4591,Y 35.991,Z 144,A 159.8007,B 24.8105,C -1.5262,E1 24.7009,E2 286.6457} C_DIS
LIN {X -122.1763,Y 40.1332,Z 144,A 157.9285,B 24.81,C -1.535,E1 24.7025,E2 288.5075} C_DIS
LIN {X -120.6516,Y 44.5091,Z 144,A 155.6282,B 24.8103,C -1.5308,E1 24.7046,E2 290.8311} C_DIS
LIN {X -119.3426,Y 47.9043,Z 144,A 154.1706,B 24.8095,C -1.5434,E1 24.7061,E2 292.2669} C_DIS
LIN {X -117.7132,Y 51.7846,Z 144,A 152.1694,B 24.8095,C -1.5434,E1 24.7083,E2 294.2791} C_DIS
LIN {X -116.1731,Y 55.1483,Z 144,A 150.54,B 24.8092,C -1.5493,E1 24.7102,E2 295.9032} C_DIS
LIN {X -114.7003,Y 58.1491,Z 144,A 149.0365,B 24.8089,C -1.5532,E1 24.7121,E2 297.4056} C_DIS
LIN {X -113.062,Y 61.2783,Z 144,A 147.3296,B 24.809,C -1.5518,E1 24.7144,E2 299.125} C_DIS
LIN {X -110.7451,Y 65.3721,Z 144,A 145.2502,B 24.8086,C -1.5587,E1 24.7172,E2 301.1988} C_DIS
LIN {X -108.494,Y 69.0441,Z 144,A 143.2899,B 24.8084,C -1.5624,E1 24.7201,E2 303.1603} C_DIS
LIN {X -106.0206,Y 72.7842,Z 144,A 141.3171,B 24.808,C -1.5692,E1 24.7232,E2 305.1267} C_DIS
LIN {X -103.429,Y 76.4231,Z 144,A 139.3314,B 24.8077,C -1.5749,E1 24.7265,E2 307.1084} C_DIS
LIN {X -99.3129,Y 81.7009,Z 144,A 135.8196,B 24.8086,C -1.5588,E1 24.7327,E2 310.6754} C_DIS
LIN {X -96.3455,Y 85.179,Z 144,A 134.4875,B 24.8064,C -1.5964,E1 24.735,E2 311.9236} C_DIS
LIN {X -92.2912,Y 89.556,Z 144,A 131.8251,B 24.806,C -1.6029,E1 24.7401,E2 314.5821} C_DIS
LIN {X -87.6182,Y 94.1327,Z 144,A 128.7067,B 24.8061,C -1.6004,E1 24.7463,E2 317.7194} C_DIS
LIN {X -84.7115,Y 96.757,Z 144,A 126.8794,B 24.8061,C -1.6007,E1 24.7502,E2 319.5535} C_DIS
LIN {X -78.9682,Y 101.4988,Z 144,A 123.5846,B 24.8056,C -1.6091,E1 24.7573,E2 322.8404} C_DIS
LIN {X -75.9322,Y 103.7896,Z 144,A 121.6034,B 24.8062,C -1.5994,E1 24.7618,E2 324.8519} C_DIS
LIN {X -73.085,Y 105.8138,Z 144,A 120.0609,B 24.806,C -1.6032,E1 24.7653,E2 326.3907} C_DIS
LIN {X -70.2671,Y 107.7057,Z 144,A 118.7871,B 24.8051,C -1.6173,E1 24.7682,E2 327.6351} C_DIS
LIN {X -66.6534,Y 109.9784,Z 144,A 116.9226,B 24.8048,C -1.6226,E1 24.7727,E2 329.4926} C_DIS
LIN {X -63.2113,Y 111.9925,Z 144,A 115.0992,B 24.8048,C -1.6237,E1 24.7771,E2 331.319} C_DIS
LIN {X -59.8435,Y 113.8252,Z 144,A 113.4775,B 24.8043,C -1.6307,E1 24.781,E2 332.9285} C_DIS
LIN {X -56.8212,Y 115.3637,Z 144,A 111.963,B 24.8041,C -1.633,E1 24.7848,E2 334.4415} C_DIS
LIN {X -53.7371,Y 116.8325,Z 144,A 110.4149,B 24.8041,C -1.6342,E1 24.7887,E2 335.9907} C_DIS
LIN {X -50.754,Y 118.1591,Z 144,A 108.8683,B 24.8042,C -1.632,E1 24.7927,E2 337.5461} C_DIS
LIN {X -46.6429,Y 119.8411,Z 144,A 106.2679,B 24.8058,C -1.6056,E1 24.7997,E2 340.2153} C_DIS
LIN {X -41.6372,Y 121.672,Z 144,A 104.5244,B 24.8038,C -1.6383,E1 24.8041,E2 341.8842} C_DIS
LIN {X -38.9065,Y 122.5716,Z 144,A 103.0816,B 24.8042,C -1.6321,E1 24.8079,E2 343.3443} C_DIS
LIN {X -34.6044,Y 123.8548,Z 144,A 101.3014,B 24.8034,C -1.6448,E1 24.8126,E2 345.0972} C_DIS
LIN {X -30.6824,Y 124.8855,Z 144,A 99.4372,B 24.8034,C -1.6438,E1 24.8177,E2 346.9664} C_DIS
LIN {X -26.6933,Y 125.7981,Z 144,A 97.5564,B 24.8035,C -1.6427,E1 24.8228,E2 348.8523} C_DIS
LIN {X -22.7023,Y 126.5785,Z 144,A 95.8637,B 24.8031,C -1.6499,E1 24.8274,E2 350.5296} C_DIS
LIN {X -19.0517,Y 127.1808,Z 144,A 94.0678,B 24.8035,C -1.6439,E1 24.8324,E2 352.3413} C_DIS
LIN {X -14.5127,Y 127.7789,Z 144,A 92.0746,B 24.8033,C -1.6474,E1 24.8379,E2 354.3278} C_DIS
LIN {X -7.7048,Y 128.3676,Z 144,A 89.2475,B 24.8025,C -1.6593,E1 24.8457,E2 357.1277} C_DIS
LIN {X -0.7809,Y 128.5962,Z 144,A 85.0896,B 24.8056,C -1.6085,E1 24.8577,E2 361.4069} C_DIS
LIN {X 5.7033,Y 128.4738,Z 144,A 83.1991,B 24.8027,C -1.6569,E1 24.8626,E2 363.1816} C_DIS
LIN {X 10.6594,Y 128.156,Z 144,A 80.9399,B 24.8028,C -1.6546,E1 24.869,E2 365.4453} C_DIS
LIN {X 14.0315,Y 127.8309,Z 144,A 79.347,B 24.8031,C -1.6503,E1 24.8734,E2 367.0475} C_DIS
LIN {X 18.067,Y 127.3229,Z 144,A 77.6093,B 24.8029,C -1.6535,E1 24.8782,E2 368.776} C_DIS
LIN {X 21.9358,Y 126.7157,Z 144,A 75.7337,B 24.8033,C -1.6464,E1 24.8834,E2 370.6665} C_DIS
LIN {X 25.4754,Y 126.0497,Z 144,A 74.2806,B 24.8029,C -1.6532,E1 24.8873,E2 372.1017} C_DIS
LIN {X 28.5606,Y 125.3866,Z 144,A 72.8699,B 24.8029,C -1.6523,E1 24.8912,E2 373.5129} C_DIS
LIN {X 31.9458,Y 124.5675,Z 144,A 71.2002,B 24.8034,C -1.6455,E1 24.8957,E2 375.1961} C_DIS
LIN {X 35.789,Y 123.5182,Z 144,A 69.5768,B 24.803,C -1.6517,E1 24.9,E2 376.802} C_DIS
LIN {X 38.6868,Y 122.6418,Z 144,A 68.0056,B 24.8037,C -1.6396,E1 24.9043,E2 378.3991} C_DIS
LIN {X 43.2689,Y 121.1008,Z 144,A 66.0119,B 24.8034,C -1.6457,E1 24.9095,E2 380.3743} C_DIS
LIN {X 46.5808,Y 119.8653,Z 144,A 64.5485,B 24.8031,C -1.6497,E1 24.9133,E2 381.825} C_DIS
LIN {X 50.672,Y 118.1945,Z 144,A 62.4679,B 24.8036,C -1.642,E1 24.9187,E2 383.9191} C_DIS
LIN {X 54.713,Y 116.3811,Z 144,A 60.4529,B 24.8039,C -1.6375,E1 24.9238,E2 385.9396} C_DIS
LIN {X 58.064,Y 114.7436,Z 144,A 58.8834,B 24.8037,C -1.6401,E1 24.9277,E2 387.4988} C_DIS
LIN {X 61.1034,Y 113.1564,Z 144,A 57.2478,B 24.8042,C -1.6325,E1 24.9318,E2 389.1478} C_DIS
LIN {X 64.8727,Y 111.0385,Z 144,A 55.4104,B 24.8041,C -1.6342,E1 24.9362,E2 390.9757} C_DIS
LIN {X 68.2744,Y 108.9802,Z 144,A 53.535,B 24.8046,C -1.6262,E1 24.9407,E2 392.8642} C_DIS
LIN {X 72.2206,Y 106.4055,Z 144,A 51.5003,B 24.8046,C -1.626,E1 24.9454,E2 394.8925} C_DIS
LIN {X 75.8156,Y 103.8753,Z 144,A 49.5119,B 24.8049,C -1.621,E1 24.95,E2 396.8857} C_DIS
LIN {X 79.1253,Y 101.3768,Z 144,A 47.6478,B 24.8051,C -1.6168,E1 24.9541,E2 398.753} C_DIS
LIN {X 82.617,Y 98.5513,Z 144,A 45.7124,B 24.8051,C -1.6163,E1 24.9583,E2 400.6821} C_DIS
LIN {X 85.9427,Y 95.665,Z 144,A 43.7477,B 24.8054,C -1.6122,E1 24.9624,E2 402.6487} C_DIS
LIN {X 89.1009,Y 92.7311,Z 144,A 41.8221,B 24.8057,C -1.6078,E1 24.9663,E2 404.5767} C_DIS
LIN {X 92.1551,Y 89.6966,Z 144,A 39.8941,B 24.806,C -1.6031,E1 24.9701,E2 406.5075} C_DIS
LIN {X 94.7798,Y 86.9179,Z 144,A 38.1885,B 24.8062,C -1.5991,E1 24.9733,E2 408.2152} C_DIS
LIN {X 97.7255,Y 83.593,Z 144,A 36.2209,B 24.8065,C -1.5951,E1 24.9769,E2 410.1835} C_DIS
LIN {X 100.912,Y 79.7171,Z 144,A 34.0689,B 24.8065,C -1.5939,E1 24.9807,E2 412.328} C_DIS
LIN {X 103.3383,Y 76.5455,Z 144,A 32.3101,B 24.8067,C -1.5905,E1 24.9837,E2 414.0865} C_DIS
LIN {X 105.7405,Y 73.1912,Z 144,A 30.4257,B 24.8072,C -1.5834,E1 24.9867,E2 415.9785} C_DIS
LIN {X 108.1309,Y 69.6114,Z 144,A 28.6182,B 24.8072,C -1.5841,E1 24.9895,E2 417.7753} C_DIS
LIN {X 110.3324,Y 66.0663,Z 144,A 26.7076,B 24.8076,C -1.5764,E1 24.9922,E2 419.6944} C_DIS
LIN {X 112.3967,Y 62.4896,Z 144,A 24.8473,B 24.8079,C -1.5702,E1 24.9948,E2 421.5596} C_DIS
LIN {X 114.4836,Y 58.5746,Z 144,A 23.0492,B 24.8077,C -1.574,E1 24.9971,E2 423.3392} C_DIS
LIN {X 115.9468,Y 55.6221,Z 144,A 21.5442,B 24.8081,C -1.5679,E1 24.999,E2 424.8505} C_DIS
LIN {X 117.3564,Y 52.5825,Z 144,A 20.114,B 24.8081,C -1.5668,E1 25.0006,E2 426.2755} C_DIS
LIN {X 119.4447,Y 47.651,Z 144,A 17.5388,B 24.8091,C -1.5498,E1 25.0034,E2 428.8766} C_DIS
LIN {X 120.8895,Y 43.8549,Z 144,A 15.9089,B 24.8089,C -1.5538,E1 25.005,E2 430.488} C_DIS
LIN {X 121.9572,Y 40.7913,Z 144,A 14.2047,B 24.81,C -1.5359,E1 25.0066,E2 432.225} C_DIS
LIN {X 123.3777,Y 36.2689,Z 144,A 12.3677,B 24.8095,C -1.5437,E1 25.008,E2 434.0329} C_DIS
LIN {X 124.243,Y 33.1838,Z 144,A 10.9282,B 24.8098,C -1.5387,E1 25.0091,E2 435.476} C_DIS
LIN {X 125.0438,Y 30.0256,Z 144,A 9.4646,B 24.8101,C -1.5335,E1 25.0101,E2 436.9434} C_DIS
LIN {X 125.9386,Y 26.0215,Z 144,A 7.6118,B 24.8105,C -1.5264,E1 25.0112,E2 438.8023} C_DIS
LIN {X 126.6072,Y 22.5419,Z 144,A 6.0651,B 24.8107,C -1.523,E1 25.012,E2 440.3478} C_DIS
LIN {X 127.2705,Y 18.4341,Z 144,A 4.2346,B 24.811,C -1.5183,E1 25.0127,E2 442.1787} C_DIS
LIN {X 127.7625,Y 14.65,Z 144,A 2.4746,B 24.8115,C -1.5096,E1 25.0133,E2 443.9488} C_DIS
LIN {X 128.324,Y 8.4125,Z 144,A -0.0766,B 24.8113,C -1.5131,E1 25.0139,E2 446.4765} C_DIS
LIN {X 128.5061,Y 4.876,Z 144,A -2.1537,B 24.8131,C -1.4816,E1 25.0142,E2 448.6157} C_DIS
LIN {X 128.5945,Y 1.1871,Z 144,A -3.401,B 24.8122,C -1.497,E1 25.0142,E2 449.8189} C_DIS
LIN {X 128.5821,Y -2.058,Z 144,A -4.8976,B 24.8126,C -1.4896,E1 25.0142,E2 451.3241} C_DIS
LIN {X 128.5042,Y -4.9232,Z 144,A -6.8129,B 24.8147,C -1.4519,E1 25.014,E2 453.3174} C_DIS
LIN {X 128.1945,Y -10.2026,Z 144,A -8.4871,B 24.8131,C -1.4799,E1 25.0137,E2 454.9153} C_DIS
LIN {X 127.8984,Y -13.4043,Z 144,A -10.3168,B 24.8146,C -1.4543,E1 25.0131,E2 456.7948} C_DIS
LIN {X 127.4255,Y -17.3376,Z 144,A -12.0628,B 24.8148,C -1.4494,E1 25.0125,E2 458.5419} C_DIS
LIN {X 126.8573,Y -21.0887,Z 144,A -13.2806,B 24.8138,C -1.4688,E1 25.0119,E2 459.7066} C_DIS
LIN {X 126.3049,Y -24.1782,Z 144,A -14.7235,B 24.8141,C -1.4618,E1 25.0112,E2 461.1575} C_DIS
LIN {X 125.4808,Y -28.1479,Z 144,A -16.5123,B 24.8144,C -1.4569,E1 25.0101,E2 462.9476} C_DIS
LIN {X 124.6784,Y -31.5087,Z 144,A -18.0239,B 24.8146,C -1.4533,E1 25.0091,E2 464.4587} C_DIS
LIN {X 123.8124,Y -34.7562,Z 144,A -19.471,B 24.8147,C -1.4512,E1 25.0081,E2 465.9026} C_DIS
LIN {X 122.6898,Y -38.5367,Z 144,A -21.3024,B 24.8153,C -1.4416,E1 25.0066,E2 467.7463} C_DIS
LIN {X 121.8239,Y -41.1918,Z 144,A -22.8517,B 24.8163,C -1.4215,E1 25.0052,E2 469.3342} C_DIS
LIN {X 120.6453,Y -44.5258,Z 144,A -24.1065,B 24.8157,C -1.4334,E1 25.004,E2 470.5538} C_DIS
LIN {X 119.368,Y -47.8414,Z 144,A -25.6193,B 24.8157,C -1.4321,E1 25.0025,E2 472.0611} C_DIS
LIN {X 118.3234,Y -50.374,Z 144,A -27.4295,B 24.8176,C -1.3973,E1 25.0004,E2 473.9439} C_DIS
LIN {X 116.4092,Y -54.6525,Z 144,A -29.0484,B 24.8167,C -1.4155,E1 24.9986,E2 475.511} C_DIS
LIN {X 114.7155,Y -58.1193,Z 144,A -30.6556,B 24.8167,C -1.4162,E1 24.9966,E2 477.1079} C_DIS
LIN {X 112.9884,Y -61.4131,Z 144,A -32.3484,B 24.817,C -1.4092,E1 24.9943,E2 478.8081} C_DIS
LIN {X 110.8116,Y -65.259,Z 144,A -34.1618,B 24.8169,C -1.4116,E1 24.9918,E2 480.6065} C_DIS
LIN {X 107.9844,Y -69.838,Z 144,A -36.6186,B 24.8174,C -1.4015,E1 24.9882,E2 483.0748} C_DIS
LIN {X 105.8431,Y -73.0424,Z 144,A -38.4942,B 24.8181,C -1.3883,E1 24.9852,E2 484.9724} C_DIS
LIN {X 102.9899,Y -77.0134,Z 144,A -40.5407,B 24.8181,C -1.3891,E1 24.9818,E2 487.0069} C_DIS
LIN {X 100.4812,Y -80.259,Z 144,A -42.4442,B 24.8185,C -1.3802,E1 24.9785,E2 488.9227} C_DIS
LIN {X 97.4211,Y -83.9466,Z 144,A -44.5075,B 24.8186,C -1.3782,E1 24.9748,E2 490.981} C_DIS
LIN {X 94.5389,Y -87.18,Z 144,A -46.3573,B 24.8186,C -1.3774,E1 24.9714,E2 492.8246} C_DIS
LIN {X 91.6855,Y -90.176,Z 144,A -48.1448,B 24.8188,C -1.3757,E1 24.9679,E2 494.6085} C_DIS
LIN {X 88.962,Y -92.8639,Z 144,A -49.913,B 24.8192,C -1.3681,E1 24.9644,E2 496.387} C_DIS
LIN {X 86.1764,Y -95.4549,Z 144,A -51.6498,B 24.8195,C -1.3619,E1 24.9608,E2 498.1316} C_DIS
LIN {X 82.9214,Y -98.2959,Z 144,A -53.5859,B 24.8197,C -1.3569,E1 24.9566,E2 500.072} C_DIS
LIN {X 79.1176,Y -101.3829,Z 144,A -55.758,B 24.82,C -1.3525,E1 24.9519,E2 502.2462} C_DIS
LIN {X 75.6936,Y -103.9638,Z 144,A -57.6586,B 24.8201,C -1.349,E1 24.9476,E2 504.1484} C_DIS
LIN {X 71.9381,Y -106.5967,Z 144,A -59.6211,B 24.8201,C -1.349,E1 24.9431,E2 506.1042} C_DIS
LIN {X 68.3668,Y -108.922,Z 144,A -61.6045,B 24.8206,C -1.3408,E1 24.9384,E2 508.1004} C_DIS
LIN {X 65.5626,Y -110.6326,Z 144,A -62.8734,B 24.8202,C -1.3481,E1 24.9355,E2 509.3482} C_DIS
LIN {X 60.9427,Y -113.2427,Z 144,A -65.7065,B 24.8216,C -1.3198,E1 24.9284,E2 512.2402} C_DIS
LIN {X 57.5408,Y -115.0088,Z 144,A -67.114,B 24.821,C -1.3322,E1 24.925,E2 513.6142} C_DIS
LIN {X 54.2383,Y -116.6007,Z 144,A -68.6246,B 24.8208,C -1.3359,E1 24.9212,E2 515.1121} C_DIS
LIN {X 49.6204,Y -118.6392,Z 144,A -70.849,B 24.8209,C -1.3337,E1 24.9155,E2 517.3363} C_DIS
LIN {X 46.578,Y -119.8663,Z 144,A -72.3356,B 24.8211,C -1.3304,E1 24.9116,E2 518.8275} C_DIS
LIN {X 42.9058,Y -121.2317,Z 144,A -74.1518,B 24.8214,C -1.3244,E1 24.9068,E2 520.6541} C_DIS
LIN {X 38.4011,Y -122.7331,Z 144,A -76.3116,B 24.8216,C -1.3195,E1 24.9011,E2 522.8214} C_DIS
LIN {X 34.6191,Y -123.8507,Z 144,A -77.8734,B 24.8212,C -1.3275,E1 24.8969,E2 524.3617} C_DIS
LIN {X 31.708,Y -124.6278,Z 144,A -79.2571,B 24.8214,C -1.324,E1 24.8932,E2 525.7515} C_DIS
LIN {X 28.322,Y -125.4411,Z 144,A -80.901,B 24.8217,C -1.3178,E1 24.8887,E2 527.4078} C_DIS
LIN {X 24.3637,Y -126.2694,Z 144,A -82.6239,B 24.8216,C -1.3202,E1 24.884,E2 529.1229} C_DIS
LIN {X 21.1333,Y -126.8499,Z 144,A -84.0623,B 24.8216,C -1.3202,E1 24.88,E2 530.5597} C_DIS
LIN {X 11.6801,Y -128.0683,Z 144,A -88.4217,B 24.822,C -1.3119,E1 24.8679,E2 534.9357} C_DIS
LIN {X 7.4997,Y -128.3802,Z 144,A -90.4457,B 24.8224,C -1.3033,E1 24.8622,E2 536.9793} C_DIS
LIN {X 1.582,Y -128.59,Z 144,A -93.1951,B 24.8227,C -1.2969,E1 24.8545,E2 539.7434} C_DIS
LIN {X 1.582,Y -128.59,Z 144,A -93.1951,B 24.8227,C -1.2969,E1 24.8545,E2 539.7434} C_DIS
Enddeposition()
LIN {X 0.9095,Y -127.6076,Z 144,A -92.3742,B 24.0822,C -1.2175,E1 24.1132,E2 539.0159} C_DIS
Startdeposition()
$VEL.CP = VEL_PRINT
LIN {X 4.3825,Y -127.5618,Z 144,A -89.8722,B 24.08,C -1.2636,E1 24.1205,E2 536.4014} C_DIS
LIN {X 9.9836,Y -127.2465,Z 144,A -88.0496,B 24.0816,C -1.2305,E1 24.1254,E2 534.6607} C_DIS
LIN {X 15.2731,Y -126.7186,Z 144,A -85.2917,B 24.0807,C -1.2502,E1 24.1331,E2 531.8567} C_DIS
LIN {X 19.2456,Y -126.1765,Z 144,A -83.9332,B 24.0817,C -1.2297,E1 24.1367,E2 530.5496} C_DIS
LIN {X 22.6655,Y -125.607,Z 144,A -82.4452,B 24.0817,C -1.2276,E1 24.1408,E2 529.0685} C_DIS
LIN {X 26.1567,Y -124.9286,Z 144,A -80.7539,B 24.0815,C -1.2336,E1 24.1455,E2 527.3646} C_DIS
LIN {X 29.7854,Y -124.1114,Z 144,A -79.1489,B 24.0815,C -1.2321,E1 24.1498,E2 525.7657} C_DIS
LIN {X 33.0725,Y -123.2762,Z 144,A -77.6088,B 24.0815,C -1.2345,E1 24.154,E2 524.2221} C_DIS
LIN {X 36.9544,Y -122.1692,Z 144,A -75.8407,B 24.0815,C -1.2344,E1 24.1587,E2 522.4575} C_DIS
LIN {X 43.9157,Y -119.8441,Z 144,A -72.5693,B 24.0813,C -1.2373,E1 24.1674,E2 519.1856} C_DIS
LIN {X 46.9728,Y -118.6799,Z 144,A -70.1512,B 24.0788,C -1.287,E1 24.174,E2 516.6516} C_DIS
LIN {X 52.7182,Y -116.241,Z 144,A -68.316,B 24.081,C -1.2427,E1 24.1784,E2 514.9297} C_DIS
LIN {X 55.2425,Y -115.0611,Z 144,A -66.9882,B 24.0807,C -1.2485,E1 24.1817,E2 513.5911} C_DIS
LIN {X 59.1884,Y -113.0818,Z 144,A -65.1556,B 24.081,C -1.2444,E1 24.1862,E2 511.7738} C_DIS
LIN {X 63.9147,Y -110.4814,Z 144,A -62.7796,B 24.0809,C -1.2464,E1 24.1921,E2 509.4001} C_DIS
LIN {X 66.6091,Y -108.8782,Z 144,A -61.1948,B 24.0803,C -1.2579,E1 24.1959,E2 507.7923} C_DIS
LIN {X 71.0803,Y -106.0135,Z 144,A -59.0245,B 24.0806,C -1.2519,E1 24.2009,E2 505.6442} C_DIS
LIN {X 73.5356,Y -104.3251,Z 144,A -57.4474,B 24.0799,C -1.2667,E1 24.2046,E2 504.0366} C_DIS
LIN {X 77.1787,Y -101.6602,Z 144,A -54.9492,B 24.0784,C -1.295,E1 24.2103,E2 501.4786} C_DIS
LIN {X 80.7159,Y -98.8745,Z 144,A -53.2605,B 24.0791,C -1.2826,E1 24.2139,E2 499.827} C_DIS
LIN {X 84.6487,Y -95.5293,Z 144,A -51.1134,B 24.0792,C -1.2792,E1 24.2184,E2 497.6969} C_DIS
LIN {X 87.7414,Y -92.6969,Z 144,A -49.0161,B 24.0785,C -1.2947,E1 24.2227,E2 495.5708} C_DIS
LIN {X 90.0619,Y -90.4438,Z 144,A -47.597,B 24.0784,C -1.2966,E1 24.2255,E2 494.1532} C_DIS
LIN {X 93.1491,Y -87.2616,Z 144,A -45.7726,B 24.0785,C -1.2931,E1 24.229,E2 492.3456} C_DIS
LIN {X 96.1531,Y -83.9393,Z 144,A -43.5255,B 24.0777,C -1.3104,E1 24.2332,E2 490.0668} C_DIS
LIN {X 98.4841,Y -81.1922,Z 144,A -41.5756,B 24.0765,C -1.3319,E1 24.2367,E2 488.0739} C_DIS
LIN {X 101.7639,Y -77.0413,Z 144,A -39.8384,B 24.0779,C -1.3055,E1 24.2396,E2 486.4095} C_DIS
LIN {X 104.4154,Y -73.4076,Z 144,A -37.6603,B 24.0772,C -1.3193,E1 24.2431,E2 484.2089} C_DIS
LIN {X 106.4892,Y -70.3656,Z 144,A -36.1866,B 24.0774,C -1.3148,E1 24.2454,E2 482.7538} C_DIS
LIN {X 109.1334,Y -66.1902,Z 144,A -34.0493,B 24.0774,C -1.317,E1 24.2485,E2 480.6224} C_DIS
LIN {X 111.0756,Y -62.8775,Z 144,A -32.2411,B 24.0768,C -1.3264,E1 24.251,E2 478.8011} C_DIS
LIN {X 113.0938,Y -59.1656,Z 144,A -30.4623,B 24.0768,C -1.3261,E1 24.2534,E2 477.0329} C_DIS
LIN {X 114.9954,Y -55.3801,Z 144,A -28.5591,B 24.0765,C -1.3319,E1 24.2557,E2 475.1261} C_DIS
LIN {X 118.3855,Y -47.7034,Z 144,A -24.8849,B 24.0762,C -1.3386,E1 24.2598,E2 471.4564} C_DIS
LIN {X 119.387,Y -45.1405,Z 144,A -22.9474,B 24.0741,C -1.3788,E1 24.2618,E2 469.4321} C_DIS
LIN {X 121.0805,Y -40.3767,Z 144,A -21.6843,B 24.0764,C -1.334,E1 24.2628,E2 468.2857} C_DIS
LIN {X 122.6777,Y -35.2334,Z 144,A -19.0282,B 24.0754,C -1.3539,E1 24.265,E2 465.5969} C_DIS
LIN {X 123.8054,Y -31.0345,Z 144,A -16.9474,B 24.0747,C -1.3668,E1 24.2665,E2 463.4971} C_DIS
LIN {X 124.7841,Y -26.8281,Z 144,A -15.0563,B 24.0745,C -1.3706,E1 24.2677,E2 461.6081} C_DIS
LIN {X 125.5743,Y -22.8482,Z 144,A -13.198,B 24.0741,C -1.3784,E1 24.2686,E2 459.7421} C_DIS
LIN {X 126.2737,Y -18.6031,Z 144,A -11.4161,B 24.0741,C -1.377,E1 24.2694,E2 457.9745} C_DIS
LIN {X 126.9627,Y -13.1006,Z 144,A -8.9888,B 24.0739,C -1.3819,E1 24.2702,E2 455.5502} C_DIS
LIN {X 127.202,Y -10.5146,Z 144,A -7.693,B 24.0733,C -1.3924,E1 24.2705,E2 454.2368} C_DIS
LIN {X 127.5613,Y -4.3962,Z 144,A -4.4009,B 24.0713,C -1.4295,E1 24.2709,E2 450.8749} C_DIS
LIN {X 127.637,Y 0.4244,Z 144,A -2.809,B 24.0725,C -1.4068,E1 24.2709,E2 449.3479} C_DIS
LIN {X 127.4207,Y 7.4173,Z 144,A 0.0856,B 24.0727,C -1.4044,E1 24.2707,E2 446.4773} C_DIS
LIN {X 127.2128,Y 10.3865,Z 144,A 1.652,B 24.0718,C -1.4205,E1 24.2703,E2 444.8811} C_DIS
LIN {X 126.8481,Y 14.1657,Z 144,A 3.3858,B 24.0714,C -1.4276,E1 24.2698,E2 443.141} C_DIS
LIN {X 126.3446,Y 18.107,Z 144,A 5.0187,B 24.0715,C -1.4255,E1 24.2692,E2 441.5231} C_DIS
LIN {X 125.7987,Y 21.5838,Z 144,A 6.7241,B 24.0709,C -1.437,E1 24.2684,E2 439.8001} C_DIS
LIN {X 125.0711,Y 25.4562,Z 144,A 8.4005,B 24.0709,C -1.4379,E1 24.2675,E2 438.1318} C_DIS
LIN {X 124.1577,Y 29.5934,Z 144,A 10.2938,B 24.0705,C -1.4434,E1 24.2663,E2 436.2365} C_DIS
LIN {X 123.3,Y 32.9834,Z 144,A 11.8205,B 24.0704,C -1.4461,E1 24.2653,E2 434.7124} C_DIS
LIN {X 122.3863,Y 36.2288,Z 144,A 13.2915,B 24.0702,C -1.4486,E1 24.2641,E2 433.2442} C_DIS
LIN {X 120.3175,Y 42.6026,Z 144,A 16.261,B 24.0698,C -1.4556,E1 24.2615,E2 430.2748} C_DIS
LIN {X 117.3273,Y 50.2518,Z 144,A 19.8075,B 24.0696,C -1.4593,E1 24.2579,E2 426.7397} C_DIS
LIN {X 115.8001,Y 53.6758,Z 144,A 21.6293,B 24.0689,C -1.4713,E1 24.2558,E2 424.8992} C_DIS
LIN {X 114.4871,Y 56.4219,Z 144,A 23.0684,B 24.0685,C -1.4789,E1 24.254,E2 423.4496} C_DIS
LIN {X 112.5885,Y 60.1262,Z 144,A 24.9797,B 24.0681,C -1.4862,E1 24.2515,E2 421.5309} C_DIS
LIN {X 110.3787,Y 64.0921,Z 144,A 27.4076,B 24.0666,C -1.5117,E1 24.2481,E2 419.054} C_DIS
LIN {X 108.1362,Y 67.808,Z 144,A 28.9538,B 24.0675,C -1.4964,E1 24.2458,E2 417.5532} C_DIS
LIN {X 105.7284,Y 71.5034,Z 144,A 30.9031,B 24.0672,C -1.5,E1 24.2428,E2 415.6051} C_DIS
LIN {X 103.3351,Y 74.9205,Z 144,A 32.73,B 24.0672,C -1.5025,E1 24.2399,E2 413.7816} C_DIS
LIN {X 100.652,Y 78.4891,Z 144,A 34.9955,B 24.066,C -1.5206,E1 24.236,E2 411.4829} C_DIS
LIN {X 98.5068,Y 81.1648,Z 144,A 36.1783,B 24.0669,C -1.5063,E1 24.2339,E2 410.3408} C_DIS
LIN {X 95.9218,Y 84.2043,Z 144,A 38.0699,B 24.0663,C -1.5155,E1 24.2304,E2 408.4355} C_DIS
LIN {X 92.7587,Y 87.6758,Z 144,A 39.8951,B 24.0669,C -1.5061,E1 24.2271,E2 406.6417} C_DIS
LIN {X 90.7031,Y 89.801,Z 144,A 41.467,B 24.066,C -1.5213,E1 24.2239,E2 405.0398} C_DIS
LIN {X 87.7713,Y 92.6686,Z 144,A 43.3271,B 24.0657,C -1.5261,E1 24.2202,E2 403.1759} C_DIS
LIN {X 84.3924,Y 95.7558,Z 144,A 45.3392,B 24.0656,C -1.5282,E1 24.216,E2 401.1671} C_DIS
LIN {X 81.1673,Y 98.5047,Z 144,A 47.2116,B 24.0654,C -1.5304,E1 24.212,E2 399.2969} C_DIS
LIN {X 77.9813,Y 101.0456,Z 144,A 48.9791,B 24.0654,C -1.5308,E1 24.2081,E2 397.5353} C_DIS
LIN {X 74.8433,Y 103.391,Z 144,A 50.806,B 24.065,C -1.5373,E1 24.204,E2 395.6993} C_DIS
LIN {X 69.7717,Y 106.8795,Z 144,A 53.5922,B 24.0647,C -1.543,E1 24.1975,E2 392.9088} C_DIS
LIN {X 65.9347,Y 109.2879,Z 144,A 55.6311,B 24.0645,C -1.5464,E1 24.1927,E2 390.8684} C_DIS
LIN {X 62.5194,Y 111.2769,Z 144,A 57.332,B 24.0645,C -1.5454,E1 24.1886,E2 389.1753} C_DIS
LIN {X 58.9781,Y 113.1922,Z 144,A 59.0809,B 24.0645,C -1.545,E1 24.1843,E2 387.4325} C_DIS
LIN {X 54.3104,Y 115.5064,Z 144,A 61.3799,B 24.0645,C -1.5459,E1 24.1785,E2 385.1376} C_DIS
LIN {X 50.3279,Y 117.2944,Z 144,A 63.3411,B 24.0644,C -1.5483,E1 24.1735,E2 383.1756} C_DIS
LIN {X 44.5679,Y 119.6014,Z 144,A 65.9344,B 24.0648,C -1.5418,E1 24.1669,E2 380.6042} C_DIS
LIN {X 41.9953,Y 120.5288,Z 144,A 67.7994,B 24.0628,C -1.5739,E1 24.1617,E2 378.6646} C_DIS
LIN {X 38.2593,Y 121.7677,Z 144,A 69.0562,B 24.0642,C -1.5505,E1 24.1585,E2 377.4675} C_DIS
LIN {X 34.3066,Y 122.9384,Z 144,A 70.9645,B 24.064,C -1.5546,E1 24.1534,E2 375.5524} C_DIS
LIN {X 30.9282,Y 123.8324,Z 144,A 72.6717,B 24.0635,C -1.5623,E1 24.1487,E2 373.8291} C_DIS
LIN {X 27.019,Y 124.7429,Z 144,A 74.3405,B 24.0639,C -1.5568,E1 24.1442,E2 372.1761} C_DIS
LIN {X 23.514,Y 125.4516,Z 144,A 76.042,B 24.0635,C -1.5621,E1 24.1395,E2 370.4636} C_DIS
LIN {X 19.403,Y 126.1521,Z 144,A 77.846,B 24.0637,C -1.5595,E1 24.1346,E2 368.6679} C_DIS
LIN {X 15.9511,Y 126.6365,Z 144,A 79.4726,B 24.0635,C -1.5628,E1 24.1301,E2 367.0346} C_DIS
LIN {X 11.8856,Y 127.0814,Z 144,A 81.2036,B 24.0638,C -1.5581,E1 24.1253,E2 365.3164} C_DIS
LIN {X 7.9872,Y 127.3856,Z 144,A 83.0266,B 24.0636,C -1.5614,E1 24.1202,E2 363.4861} C_DIS
LIN {X 4.5446,Y 127.5555,Z 144,A 85.1327,B 24.0619,C -1.588,E1 24.1141,E2 361.3155} C_DIS
LIN {X -0.2068,Y 127.6365,Z 144,A 86.5162,B 24.0642,C -1.5519,E1 24.1105,E2 360.0204} C_DIS
LIN {X -6.2161,Y 127.4843,Z 144,A 89.1439,B 24.0644,C -1.5478,E1 24.1032,E2 357.4025} C_DIS
LIN {X -10.3512,Y 127.2158,Z 144,A 91.217,B 24.0638,C -1.557,E1 24.0974,E2 355.306} C_DIS
LIN {X -13.4509,Y 126.925,Z 144,A 92.6547,B 24.0638,C -1.5582,E1 24.0934,E2 353.8646} C_DIS
LIN {X -16.6521,Y 126.5446,Z 144,A 94.0764,B 24.0638,C -1.5561,E1 24.0894,E2 352.4468} C_DIS
LIN {X -20.5053,Y 125.9786,Z 144,A 95.8833,B 24.0638,C -1.5577,E1 24.0844,E2 350.6345} C_DIS
LIN {X -23.9816,Y 125.3622,Z 144,A 97.4099,B 24.064,C -1.5537,E1 24.0803,E2 349.1159} C_DIS
LIN {X -27.8623,Y 124.5585,Z 144,A 99.3642,B 24.0636,C -1.5603,E1 24.0749,E2 347.1429} C_DIS
LIN {X -32.5259,Y 123.422,Z 144,A 101.3911,B 24.0641,C -1.5523,E1 24.0694,E2 345.1328} C_DIS
LIN {X -35.8948,Y 122.484,Z 144,A 103.6314,B 24.0623,C -1.5818,E1 24.0632,E2 342.816} C_DIS
LIN {X -40.9529,Y 120.8886,Z 144,A 105.4893,B 24.064,C -1.5545,E1 24.0585,E2 341.0216} C_DIS
LIN {X -47.2811,Y 118.5558,Z 144,A 108.3225,B 24.0648,C -1.5415,E1 24.0512,E2 338.2141} C_DIS
LIN {X -50.587,Y 117.1823,Z 144,A 109.9358,B 24.0648,C -1.5395,E1 24.047,E2 336.6019} C_DIS
LIN {X -53.5909,Y 115.8393,Z 144,A 111.4266,B 24.065,C -1.5379,E1 24.0432,E2 335.1113} C_DIS
LIN {X -56.7575,Y 114.3216,Z 144,A 113.0057,B 24.0651,C -1.5355,E1 24.0392,E2 333.5339} C_DIS
LIN {X -60.1079,Y 112.5983,Z 144,A 114.8251,B 24.065,C -1.5385,E1 24.0347,E2 331.7018} C_DIS
LIN {X -63.9055,Y 110.4867,Z 144,A 116.7871,B 24.0651,C -1.5356,E1 24.03,E2 329.741} C_DIS
LIN {X -67.8073,Y 108.1366,Z 144,A 118.866,B 24.0653,C -1.5333,E1 24.025,E2 327.661} C_DIS
LIN {X -71.6193,Y 105.6499,Z 144,A 120.7176,B 24.066,C -1.5206,E1 24.0208,E2 325.8343} C_DIS
LIN {X -75.9051,Y 102.6148,Z 144,A 122.97,B 24.0666,C -1.511,E1 24.0157,E2 323.5974} C_DIS
LIN {X -78.051,Y 100.9916,Z 144,A 124.4579,B 24.066,C -1.5211,E1 24.0123,E2 322.079} C_DIS
LIN {X -82.8619,Y 97.0834,Z 144,A 127.7806,B 24.0649,C -1.5394,E1 24.0051,E2 318.6979} C_DIS
LIN {X -86.42,Y 93.9297,Z 144,A 129.3949,B 24.0666,C -1.5108,E1 24.0019,E2 317.1472} C_DIS
LIN {X -90.9008,Y 89.6012,Z 144,A 132.0122,B 24.0675,C -1.496,E1 23.9967,E2 314.555} C_DIS
LIN {X -95.0655,Y 85.1691,Z 144,A 134.6059,B 24.0682,C -1.483,E1 23.9918,E2 311.9815} C_DIS
LIN {X -96.858,Y 83.1252,Z 144,A 136.512,B 24.0666,C -1.5105,E1 23.9882,E2 309.9985} C_DIS
LIN {X -99.2649,Y 80.2351,Z 144,A 138.111,B 24.0671,C -1.502,E1 23.9854,E2 308.4127} C_DIS
LIN {X -101.3078,Y 77.64,Z 144,A 139.3217,B 24.0681,C -1.4858,E1 23.9834,E2 307.2359} C_DIS
LIN {X -103.656,Y 74.4764,Z 144,A 141.1291,B 24.0683,C -1.4827,E1 23.9804,E2 305.4271} C_DIS
LIN {X -105.9303,Y 71.205,Z 144,A 142.9918,B 24.0683,C -1.481,E1 23.9775,E2 303.5589} C_DIS
LIN {X -108.3488,Y 67.4667,Z 144,A 144.941,B 24.0688,C -1.4731,E1 23.9746,E2 301.6189} C_DIS
LIN {X -110.5707,Y 63.7604,Z 144,A 147.2346,B 24.0682,C -1.4833,E1 23.9713,E2 299.2879} C_DIS
LIN {X -112.3828,Y 60.5091,Z 144,A 148.5284,B 24.0695,C -1.4615,E1 23.9696,E2 298.0406} C_DIS
LIN {X -113.7802,Y 57.8343,Z 144,A 149.8648,B 24.0698,C -1.4567,E1 23.9679,E2 296.7087} C_DIS
LIN {X -115.2869,Y 54.7698,Z 144,A 151.4202,B 24.07,C -1.453,E1 23.966,E2 295.1534} C_DIS
LIN {X -117.8105,Y 49.1064,Z 144,A 154.2098,B 24.0704,C -1.4448,E1 23.9629,E2 292.3682} C_DIS
LIN {X -119.0493,Y 46.0226,Z 144,A 155.7341,B 24.0706,C -1.4416,E1 23.9614,E2 290.8429} C_DIS
LIN {X -120.295,Y 42.6651,Z 144,A 157.4331,B 24.0706,C -1.4406,E1 23.9597,E2 289.1364} C_DIS
LIN {X -121.4397,Y 39.2859,Z 144,A 159.8693,B 24.0688,C -1.4728,E1 23.9576,E2 286.6061} C_DIS
LIN {X -123.2163,Y 33.2972,Z 144,A 161.6006,B 24.072,C -1.416,E1 23.9564,E2 285.0045} C_DIS
LIN {X -124.8156,Y 26.682,Z 144,A 164.7859,B 24.0723,C -1.4118,E1 23.9543,E2 281.81} C_DIS
LIN {X -125.4199,Y 23.6801,Z 144,A 166.3183,B 24.0721,C -1.4144,E1 23.9535,E2 280.2619} C_DIS
LIN {X -126.1254,Y 19.5759,Z 144,A 168.1274,B 24.0726,C -1.4056,E1 23.9527,E2 278.4631} C_DIS
LIN {X -126.6797,Y 15.599,Z 144,A 170.0351,B 24.0726,C -1.4044,E1 23.952,E2 276.5466} C_DIS
LIN {X -127.1206,Y 11.4767,Z 144,A 171.9317,B 24.0729,C -1.3999,E1 23.9515,E2 274.6493} C_DIS
LIN {X -127.4036,Y 7.6937,Z 144,A 173.5772,B 24.0734,C -1.3918,E1 23.9512,E2 273.0134} C_DIS
LIN {X -127.5836,Y 3.6464,Z 144,A 175.3707,B 24.0737,C -1.3848,E1 23.951,E2 271.226} C_DIS
LIN {X -127.6397,Y 0,Z 144,A 177.1589,B 24.0737,C -1.3861,E1 23.951,E2 269.4234} C_DIS
LIN {X -127.5768,Y -3.8906,Z 144,A 178.8678,B 24.0741,C -1.3787,E1 23.951,E2 267.7218} C_DIS
LIN {X -127.3926,Y -7.8732,Z 144,A -179.4161,B 24.0746,C -1.3697,E1 23.9513,E2 266.0172} C_DIS
LIN {X -127.0704,Y -11.9999,Z 144,A -177.5493,B 24.0749,C -1.3641,E1 23.9518,E2 264.1526} C_DIS
LIN {X -126.6952,Y -15.4691,Z 144,A -175.9128,B 24.0749,C -1.3621,E1 23.9523,E2 262.5106} C_DIS
LIN {X -126.1423,Y -19.4664,Z 144,A -174.1565,B 24.0754,C -1.3539,E1 23.953,E2 260.7638} C_DIS
LIN {X -125.5907,Y -22.7566,Z 144,A -172.6857,B 24.0757,C -1.348,E1 23.9537,E2 259.2986} C_DIS
LIN {X -124.8355,Y -26.5898,Z 144,A -170.8553,B 24.0758,C -1.3458,E1 23.9547,E2 257.4621} C_DIS
LIN {X -124.0624,Y -29.9887,Z 144,A -169.3077,B 24.0761,C -1.3402,E1 23.9557,E2 255.9189} C_DIS
LIN {X -122.6038,Y -35.4857,Z 144,A -166.9247,B 24.0769,C -1.3247,E1 23.9575,E2 253.5597} C_DIS
LIN {X -121.0646,Y -40.4245,Z 144,A -164.4813,B 24.077,C -1.323,E1 23.9595,E2 251.1058} C_DIS
LIN {X -120.0754,Y -43.2741,Z 144,A -163.0596,B 24.077,C -1.322,E1 23.9609,E2 249.6783} C_DIS
LIN {X -118.9695,Y -46.2278,Z 144,A -161.6397,B 24.0773,C -1.3179,E1 23.9623,E2 248.2601} C_DIS
LIN {X -117.7582,Y -49.2315,Z 144,A -160.1557,B 24.0774,C -1.315,E1 23.9638,E2 246.7746} C_DIS
LIN {X -116.4697,Y -52.2069,Z 144,A -158.6754,B 24.0776,C -1.3119,E1 23.9655,E2 245.2936} C_DIS
LIN {X -113.5914,Y -58.2051,Z 144,A -155.7349,B 24.0781,C -1.3013,E1 23.9691,E2 242.3626} C_DIS
LIN {X -112.1829,Y -60.8787,Z 144,A -154.249,B 24.0781,C -1.3034,E1 23.9711,E2 240.8635} C_DIS
LIN {X -110.3208,Y -64.1921,Z 144,A -152.4985,B 24.0781,C -1.3007,E1 23.9735,E2 239.1099} C_DIS
LIN {X -108.0983,Y -67.868,Z 144,A -150.6607,B 24.0786,C -1.2915,E1 23.9762,E2 237.2851} C_DIS
LIN {X -104.3324,Y -73.5254,Z 144,A -147.6099,B 24.079,C -1.2836,E1 23.981,E2 234.238} C_DIS
LIN {X -100.6567,Y -78.4829,Z 144,A -144.9907,B 24.0797,C -1.2698,E1 23.9853,E2 231.6395} C_DIS
LIN {X -97.5134,Y -82.356,Z 144,A -142.4232,B 24.0792,C -1.2794,E1 23.9899,E2 229.036} C_DIS
LIN {X -94.6698,Y -85.609,Z 144,A -140.4933,B 24.0795,C -1.2745,E1 23.9935,E2 227.1092} C_DIS
LIN {X -91.5352,Y -88.9527,Z 144,A -138.4455,B 24.0797,C -1.2695,E1 23.9974,E2 225.0644} C_DIS
LIN {X -88.4992,Y -91.9743,Z 144,A -136.4836,B 24.0798,C -1.2672,E1 24.0014,E2 223.0996} C_DIS
LIN {X -85.32,Y -94.9303,Z 144,A -134.5358,B 24.08,C -1.2632,E1 24.0054,E2 221.1535} C_DIS
LIN {X -81.9192,Y -97.88,Z 144,A -132.3889,B 24.08,C -1.2651,E1 24.01,E2 218.9933} C_DIS
LIN {X -78.6436,Y -100.5309,Z 144,A -130.6229,B 24.0804,C -1.2558,E1 24.0138,E2 217.2434} C_DIS
LIN {X -73.6569,Y -104.2396,Z 144,A -128.2168,B 24.0815,C -1.2331,E1 24.0191,E2 214.8841} C_DIS
LIN {X -69.8013,Y -106.8603,Z 144,A -125.7179,B 24.0808,C -1.2485,E1 24.025,E2 212.3388} C_DIS
LIN {X -65.7541,Y -109.3971,Z 144,A -123.6787,B 24.0811,C -1.2403,E1 24.0298,E2 210.313} C_DIS
LIN {X -62.3958,Y -111.3464,Z 144,A -121.8308,B 24.0811,C -1.2428,E1 24.0343,E2 208.4535} C_DIS
LIN {X -57.4492,Y -113.9762,Z 144,A -119.5281,B 24.0817,C -1.2295,E1 24.04,E2 206.1767} C_DIS
LIN {X -54.9352,Y -115.2079,Z 144,A -118.1578,B 24.0815,C -1.2333,E1 24.0435,E2 204.7934} C_DIS
LIN {X -51.5882,Y -116.7464,Z 144,A -115.8126,B 24.08,C -1.2641,E1 24.0497,E2 202.3667} C_DIS
LIN {X -46.9326,Y -118.6955,Z 144,A -114.1018,B 24.0814,C -1.2355,E1 24.0539,E2 200.7223} C_DIS
LIN {X -41.293,Y -120.7723,Z 144,A -111.578,B 24.0819,C -1.2248,E1 24.0605,E2 198.2194} C_DIS
LIN {X -38.6601,Y -121.6396,Z 144,A -110.2298,B 24.0817,C -1.2288,E1 24.0641,E2 196.859} C_DIS
LIN {X -34.644,Y -122.844,Z 144,A -108.3597,B 24.0817,C -1.2269,E1 24.0691,E2 194.9903} C_DIS
LIN {X -31.3082,Y -123.736,Z 144,A -106.8373,B 24.0819,C -1.2246,E1 24.0732,E2 193.4711} C_DIS
LIN {X -28.2853,Y -124.4619,Z 144,A -105.417,B 24.0819,C -1.2251,E1 24.0771,E2 192.0477} C_DIS
LIN {X -24.7696,Y -125.2108,Z 144,A -103.7336,B 24.0818,C -1.2277,E1 24.0817,E2 190.3559} C_DIS
LIN {X -20.0493,Y -126.0513,Z 144,A -101.286,B 24.0811,C -1.2412,E1 24.0886,E2 187.8727} C_DIS
LIN {X -16.5817,Y -126.5539,Z 144,A -100.1266,B 24.0821,C -1.221,E1 24.0916,E2 186.762} C_DIS
LIN {X -13.6186,Y -126.9069,Z 144,A -98.1456,B 24.0806,C -1.2518,E1 24.0974,E2 184.7042} C_DIS
LIN {X -8.9539,Y -127.3216,Z 144,A -97.0303,B 24.0829,C -1.204,E1 24.1002,E2 183.7055} C_DIS
LIN {X -2.5151,Y -127.6115,Z 144,A -93.8604,B 24.0822,C -1.2175,E1 24.1091,E2 180.5019} C_DIS
LIN {X 0.9095,Y -127.6076,Z 144,A -92.3704,B 24.0823,C -1.2159,E1 24.1132,E2 179.0158} C_DIS
Enddeposition()
LIN {X 0.9095,Y -127.6076,Z 144,A -92.3704,B 24.0823,C -1.2159,E1 24.1132,E2 179.0158} C_DIS
Startdeposition()
$VEL.CP = VEL_PRINT
LIN {X -1.0019,Y -126.6693,Z 144,A -93.5173,B 23.3579,C -1.076,E1 23.3794,E2 180.4155} C_DIS
LIN {X -7.0579,Y -126.4776,Z 144,A -96.2405,B 23.3579,C -1.0765,E1 23.3718,E2 183.1381} C_DIS
LIN {X -11.9717,Y -126.1059,Z 144,A -98.4774,B 23.3579,C -1.0762,E1 23.3656,E2 185.3766} C_DIS
LIN {X -15.4613,Y -125.7265,Z 144,A -100.0729,B 23.3579,C -1.0762,E1 23.3612,E2 186.9735} C_DIS
LIN {X -21.0669,Y -124.9088,Z 144,A -102.2331,B 23.3571,C -1.0951,E1 23.3553,E2 189.0878} C_DIS
LIN {X -23.5972,Y -124.4555,Z 144,A -103.8472,B 23.358,C -1.075,E1 23.3507,E2 190.7544} C_DIS
LIN {X -27.2086,Y -123.717,Z 144,A -105.4351,B 23.3578,C -1.0793,E1 23.3464,E2 192.3335} C_DIS
LIN {X -29.8295,Y -123.1104,Z 144,A -106.7468,B 23.3579,C -1.0757,E1 23.3428,E2 193.6562} C_DIS
LIN {X -33.8838,Y -122.0569,Z 144,A -108.6127,B 23.3579,C -1.0782,E1 23.3378,E2 195.5189} C_DIS
LIN {X -37.0348,Y -121.1377,Z 144,A -110.0984,B 23.3578,C -1.0792,E1 23.3338,E2 197.0047} C_DIS
LIN {X -40.3162,Y -120.0859,Z 144,A -112.0363,B 23.3585,C -1.0635,E1 23.3286,E2 198.9861} C_DIS
LIN {X -43.7511,Y -118.8793,Z 144,A -113.2652,B 23.3576,C -1.0836,E1 23.3255,E2 200.1669} C_DIS
LIN {X -49.6735,Y -116.5284,Z 144,A -116.1231,B 23.3574,C -1.0875,E1 23.3181,E2 203.0216} C_DIS
LIN {X -52.2222,Y -115.4082,Z 144,A -117.4158,B 23.3574,C -1.0875,E1 23.3148,E2 204.3179} C_DIS
LIN {X -54.8436,Y -114.1847,Z 144,A -118.8,B 23.3574,C -1.0857,E1 23.3113,E2 205.7103} C_DIS
LIN {X -60.0238,Y -111.5505,Z 144,A -121.5583,B 23.3576,C -1.0833,E1 23.3044,E2 208.4828} C_DIS
LIN {X -64.1257,Y -109.2441,Z 144,A -123.6934,B 23.3575,C -1.0861,E1 23.2992,E2 210.6176} C_DIS
LIN {X -66.9228,Y -107.5533,Z 144,A -125.1139,B 23.3573,C -1.0908,E1 23.2959,E2 212.0309} C_DIS
LIN {X -70.6675,Y -105.1315,Z 144,A -127.1909,B 23.3573,C -1.0914,E1 23.291,E2 214.1138} C_DIS
LIN {X -75.5439,Y -101.683,Z 144,A -129.8556,B 23.357,C -1.0977,E1 23.285,E2 216.7726} C_DIS
LIN {X -79.0747,Y -98.9624,Z 144,A -131.9645,B 23.357,C -1.0974,E1 23.2803,E2 218.8908} C_DIS
LIN {X -82.6749,Y -95.9752,Z 144,A -133.9841,B 23.3566,C -1.1056,E1 23.276,E2 220.8978} C_DIS
LIN {X -85.9145,Y -93.0867,Z 144,A -135.9841,B 23.3566,C -1.108,E1 23.2719,E2 222.9006} C_DIS
LIN {X -89.0484,Y -90.0936,Z 144,A -137.9917,B 23.3564,C -1.11,E1 23.2679,E2 224.912} C_DIS
LIN {X -92.1446,Y -86.9237,Z 144,A -139.9599,B 23.3562,C -1.116,E1 23.2641,E2 226.8742} C_DIS
LIN {X -95.1129,Y -83.666,Z 144,A -141.974,B 23.356,C -1.1196,E1 23.2603,E2 228.8888} C_DIS
LIN {X -97.8882,Y -80.4013,Z 144,A -143.9523,B 23.3559,C -1.1224,E1 23.2568,E2 230.8699} C_DIS
LIN {X -101.849,Y -75.3213,Z 144,A -146.5759,B 23.355,C -1.142,E1 23.2524,E2 233.4574} C_DIS
LIN {X -105.8983,Y -69.5123,Z 144,A -149.8098,B 23.3547,C -1.1487,E1 23.2472,E2 236.6912} C_DIS
LIN {X -107.4683,Y -67.0594,Z 144,A -151.3909,B 23.355,C -1.1409,E1 23.2448,E2 238.3009} C_DIS
LIN {X -109.8033,Y -63.1643,Z 144,A -153.6079,B 23.355,C -1.1395,E1 23.2417,E2 240.5338} C_DIS
LIN {X -111.4754,Y -60.1637,Z 144,A -155.0662,B 23.3547,C -1.1478,E1 23.2397,E2 241.9794} C_DIS
LIN {X -113.4733,Y -56.3009,Z 144,A -157.238,B 23.3548,C -1.1447,E1 23.237,E2 244.1717} C_DIS
LIN {X -114.8873,Y -53.3559,Z 144,A -158.1411,B 23.3535,C -1.1732,E1 23.236,E2 245.0077} C_DIS
LIN {X -116.4734,Y -49.8006,Z 144,A -160.1112,B 23.3537,C -1.1694,E1 23.2337,E2 246.9993} C_DIS
LIN {X -117.5027,Y -47.3183,Z 144,A -161.3936,B 23.3537,C -1.1701,E1 23.2324,E2 248.2875} C_DIS
LIN {X -118.7082,Y -44.2079,Z 144,A -162.8451,B 23.3533,C -1.177,E1 23.2309,E2 249.7304} C_DIS
LIN {X -119.691,Y -41.4727,Z 144,A -164.2423,B 23.3533,C -1.1774,E1 23.2296,E2 251.135} C_DIS
LIN {X -121.3633,Y -36.2962,Z 144,A -166.9382,B 23.3534,C -1.1749,E1 23.2274,E2 253.854} C_DIS
LIN {X -122.9131,Y -30.6368,Z 144,A -169.3432,B 23.3525,C -1.1935,E1 23.2257,E2 256.2268} C_DIS
LIN {X -123.7245,Y -27.1735,Z 144,A -171.1419,B 23.3527,C -1.1906,E1 23.2245,E2 258.0444} C_DIS
LIN {X -124.4099,Y -23.8359,Z 144,A -172.5825,B 23.3522,C -1.1996,E1 23.2238,E2 259.4713} C_DIS
LIN {X -125.0637,Y -20.1386,Z 144,A -174.411,B 23.3522,C -1.1996,E1 23.2229,E2 261.3118} C_DIS
Enddeposition()
END
